// TwinCAT 3 PLC project Fraktal_Tests
// Title: Fraktal_Tests
// Company: fraktal-automation
// Author: fraktal-automation
// ProjectVersion: 0.1.0.10
// Description: Aggregate Fraktal Core + Modules + Press Demo TcUnit gate - excluded from deployed runtime (Core 5.7).
// ProgramVersion: 3.1.4026.24
// libraries:
//   Tc2_Standard, * (Beckhoff Automation GmbH)
//   Tc2_System, * (Beckhoff Automation GmbH)
//   Tc2_Utilities, * (Beckhoff Automation GmbH)
//   Tc3_Module, * (Beckhoff Automation GmbH)
//   Fraktal_Core, 0.25.0.0 (fraktal-automation)
//   Tc2_MC2, * (Beckhoff Automation GmbH)
//   Fraktal_Modules, 0.11.0.3 (fraktal-automation)
//   TcUnit, * (www.tcunit.org)
// project tree:
//   Fraktal_Tests/ FB_ProbeWeeklyLine.TcPOU, FB_Handover_Tests.TcPOU, FB_ProbeRecipeCatalog.TcPOU, PlcTask.TcTTO (not stored), FB_Access_Tests.TcPOU, FB_AlarmLog_Tests.TcPOU (not stored), FB_Base_Tests.TcPOU, FB_ConfigurableCylinderCM_Tests.TcPOU (not stored), FB_ClampEM_Tests.TcPOU, FB_ProbeClampCycle.TcPOU, FB_ProbeClampRoot.TcPOU, FB_UnitTier_Tests.TcPOU, FB_Connector_Tests.TcPOU, FB_CylinderCM_Tests.TcPOU, FB_Decision_Tests.TcPOU, FB_Hmi_Tests.TcPOU, FB_HostEvent_Tests.TcPOU, FB_IoTopologyPublisher_Tests.TcPOU (not stored), FB_InputCM_Tests.TcPOU, FB_ManualCmd_Tests.TcPOU (not stored), FB_MultiRoot_Tests.TcPOU (not stored), FB_Oee_Tests.TcPOU (not stored), FB_PermIntlk_Tests.TcPOU (not stored), FB_PowerGroupCM_Tests.TcPOU (not stored), FB_TwoHandStartCM_Tests.TcPOU (not stored), FB_ConfigWrite_Tests.TcPOU, FB_ProbeConfigPersistence.TcPOU, FB_Shift_Tests.TcPOU, FB_LineData_Tests.TcPOU, FB_ProbeLineSource.TcPOU, FB_ProbeLineUnit.TcPOU, FB_Sha256_Tests.TcPOU, FB_ModelData_Tests.TcPOU, FB_ProbeModelUnit.TcPOU, ST_ProbeModelParCfg.TcDUT, FB_DataClass_Tests.TcPOU, FB_ConfigSet_Tests.TcPOU, FB_ConfigDurability_Tests.TcPOU, FB_ProbeConfigCM.TcPOU, FB_ProbeConfigUnit.TcPOU, FB_ProbeCM.TcPOU, FB_ProbeConnector.TcPOU (not stored), FB_ProbeRaiseChain.TcPOU, FB_ProbeUnitRaise.TcPOU, FB_SequenceRaise_Tests.TcPOU, FB_ProbeLeg.TcPOU, FB_ProbeParChain.TcPOU, FB_ProbeUnitPar.TcPOU, FB_SequencePar_Tests.TcPOU, FB_RobotConnector_Tests.TcPOU, FB_RobotCM_Tests.TcPOU, FB_AxisJog_Tests.TcPOU, FB_Separator_Tests.TcPOU, FB_Engineering_Tests.TcPOU, FB_RobotPlanner_Tests.TcPOU, FB_Separator_Tests.TcPOU, FB_Engineering_Tests.TcPOU, FB_Axis_Tests.TcPOU, FB_Separator_Tests.TcPOU, FB_Engineering_Tests.TcPOU, FB_StateFlag_Tests.TcPOU, FB_ProbeEM.TcPOU (not stored), FB_ProbeUnit.TcPOU, FB_ProbeUnitManual.TcPOU (not stored), FB_Release_Tests.TcPOU (not stored), FB_PartTrace_Tests.TcPOU (not stored), FB_Shelve_Tests.TcPOU, FB_SystemInfrastructure_Tests.TcPOU, FB_TcpDev_Tests.TcPOU (not stored), FB_Timing_Tests.TcPOU, FB_Unit_Tests.TcPOU, FB_ProbeAccessStore.TcPOU, FB_ProbeFileOps.TcPOU, F_ProbeAlarmActive.TcPOU, FB_AccessPersistence_Tests.TcPOU, FB_PlatformHealth_Tests.TcPOU, FB_PersistMedium_Tests.TcPOU, FB_LiveConfig_Tests.TcPOU, PRG_PlatformAcceptance.TcPOU, PRG_TcUnitRunner.TcPOU
// real-time tasks:
//   TASK PlcTask: cycle T#10ms, priority 20, ADS port 350

// ---- Fraktal_Tests/ST_ProbeModelParCfg.TcDUT
// §3.8a probe recipe record: the probe root's own model data.
TYPE ST_ProbeModelParCfg :
STRUCT
    SchemaVersion : UINT := 1;
    Speed         : DINT;
END_STRUCT
END_TYPE

// ---- Fraktal_Tests/FB_ProbeWeeklyLine.TcPOU
FUNCTION_BLOCK FB_ProbeWeeklyLine EXTENDS FB_LineDataV3

Cyclic();

METHOD M_ResetFixture
VAR
    i : INT;
END_VAR
    CalendarV3.SchemaVersion := 3;
    CalendarV3.UtcOffsetMin := 0;
    FOR i := 1 TO PL_Fraktal.MAX_WEEKLY_SHIFTS DO
        CalendarV3.Rows[i].StartMin := -1;
        CalendarV3.Rows[i].DurationMin := 1440;
        CalendarV3.Rows[i].ActiveDays := 0;
        CalendarV3.Rows[i].ProductionTarget := 0;
    END_FOR
END_METHOD

END_FUNCTION_BLOCK

// ---- Fraktal_Tests/FB_Handover_Tests.TcPOU
// AB-to-TC3 portable behavior, exercised in the actual IEC implementation.
FUNCTION_BLOCK FB_Handover_Tests EXTENDS TcUnit.FB_TestSuite
VAR
    _models : FB_ProbeRecipeCatalog;
    _unit : FB_ProbeModelUnit;
    _shift : FB_ProbeConfigUnit;
    _line : FB_ProbeWeeklyLine;
    _schedule : FB_ShiftSchedule;
    _calendar : ST_ShiftCalendarV3;
    _daily : ST_ShiftCalendar;
    _v2 : ST_ShiftCalendarV2;
    _loaded, _default, _a, _b : ST_ProbeModelParCfg;
    _store : FB_LocalConfigStore;
    _info : ST_ConfigSetInfo;
    _record : ST_ConfigRecord;
    _json : FB_ConfigSetJson;
    _init : BOOL;
    _done : ARRAY[1..18] OF BOOL;
    _idx : INT;
    _start, _end : DT;
    _target : UDINT;
    _i : INT;
END_VAR

IF NOT _init THEN
    _init := TRUE;
    _models.M_ResetFixture();
    _default.Speed := 1; _a.Speed := 10; _b.Speed := 20;
    _models.Register(ModelCode := '', RecipeKey := 'ProbeModel', pData := ADR(_default), Size := SIZEOF(_default));
    _models.Register(ModelCode := 'A', RecipeKey := 'ProbeModel', pData := ADR(_a), Size := SIZEOF(_a));
    _models.Register(ModelCode := 'B', RecipeKey := 'ProbeModel', pData := ADR(_b), Size := SIZEOF(_b));
    _unit.ParCfg := _default;
    _unit.Setup(Name := 'Test.Handover', Provider := _models);
    _unit();
    _unit.SetConfigStore(Store := _store);
    FOR _i := 1 TO PL_Fraktal.MAX_CONFIG_SETS DO
        IF _store.M_InfoAt(Index := 1, Info := _info) THEN _store.M_Delete(SetName := _info.SetName); END_IF
    END_FOR
    _line.M_ResetFixture();
    _line.Setup(Name := 'Test.WeeklyLine', LineId := 'handover', Role := E_LineRole.OWNER,
        Source := 0, StaleAfterMs := 0);
    _line();
    _shift.Setup(Name := 'Test.Weekly');
    _shift.SetLine(pLine := ADR(_line));
END_IF
Clone_is_inactive_and_preserves_ordinals();
Duplicate_missing_and_oversize_models_are_atomic();
Clone_rechecks_effective_read_and_write_access();
Complete_model_set_creates_without_running_load();
Current_export_is_immutable_and_uses_no_saved_slot();
Current_export_replay_and_connection_mix_are_refused();
Current_export_rechecks_permissions_and_logout();
Aborted_overwrite_preserves_the_previous_saved_set();
Daily_and_V2_migration_preserve_identity_and_disable_fifth();
Weekly_validation_rejects_overlap_wrap_and_bad_ranges();
Five_rows_select_their_own_weekday_boundaries();
Whole_calendar_transaction_is_atomic();
Off_time_production_and_empty_calendar_edits_are_preserved();
Target_edits_wait_for_boundary_and_history_is_immutable();
Clock_jumps_close_once_without_negative_history();
Manual_OEE_reset_aligns_factors_with_new_count_epoch();
Busy_creation_and_full_catalog_preserve_existing_storage();
Weekly_owner_builds_its_complete_image();

METHOD Clone_is_inactive_and_preserves_ordinals
TEST('Clone_is_inactive_and_preserves_ordinals');
IF NOT _done[1] THEN
AssertTrue(Condition := _unit.CreateModel(ModelCode := 'C', SourceIndex := 2,
    FromSet := FALSE, SetName := ''), Message := 'clone accepted');
AssertEquals_INT(Expected := 3, Actual := _unit.AvailableModelCount, Message := 'appended');
AssertEquals_STRING(Expected := 'A', Actual := _unit.AvailableModels[1].ModelCode, Message := 'ordinal A unchanged');
AssertEquals_STRING(Expected := 'B', Actual := _unit.AvailableModels[2].ModelCode, Message := 'ordinal B unchanged');
AssertEquals_DINT(Expected := 1, Actual := _unit.ParCfg.Speed, Message := 'live recipe unchanged');
AssertTrue(Condition := _models.Load(ModelCode := 'C', RecipeKey := 'ProbeModel',
    pParCfg := ADR(_loaded), Size := SIZEOF(_loaded)), Message := 'provider owns clone');
AssertEquals_DINT(Expected := 20, Actual := _loaded.Speed, Message := 'source model copied');
    _done[1] := TRUE;
END_IF
TEST_FINISHED();
END_METHOD

METHOD Duplicate_missing_and_oversize_models_are_atomic
TEST('Duplicate_missing_and_oversize_models_are_atomic');
IF NOT _done[2] THEN
AssertFalse(Condition := _unit.CreateModel(ModelCode := 'C', SourceIndex := 0, FromSet := FALSE,
    SetName := ''), Message := 'duplicate refused');
AssertFalse(Condition := _unit.CreateModel(ModelCode := 'D', SourceIndex := 99, FromSet := FALSE,
    SetName := ''), Message := 'missing source refused');
AssertFalse(Condition := _unit.CreateModel(ModelCode := 'abcdefghijklmnopqrstuvwxyzabcdefghijklmnopqrstuvwxyzabcdefghijklm',
    SourceIndex := 0, FromSet := FALSE, SetName := ''), Message := '65-byte code refused');
AssertEquals_INT(Expected := 3, Actual := _unit.AvailableModelCount, Message := 'no partial publication');
    _done[2] := TRUE;
END_IF
TEST_FINISHED();
END_METHOD

METHOD Clone_rechecks_effective_read_and_write_access
TEST('Clone_rechecks_effective_read_and_write_access');
IF NOT _done[3] THEN
_unit.M_SetConfigAccess(WriteKey := 'probe.speed', ClassId := '',
    MinReadLevel := E_AccessLevel.ENGINEER, MinWriteLevel := E_AccessLevel.NONE);
AssertFalse(Condition := _unit.CreateModel(ModelCode := 'DeniedRead', SourceIndex := 0,
    FromSet := FALSE, SetName := ''), Message := 'read denied');
_unit.M_SetConfigAccess(WriteKey := 'probe.speed', ClassId := '',
    MinReadLevel := E_AccessLevel.NONE, MinWriteLevel := E_AccessLevel.ENGINEER);
AssertFalse(Condition := _unit.CreateModel(ModelCode := 'DeniedWrite', SourceIndex := 0,
    FromSet := FALSE, SetName := ''), Message := 'write denied');
_unit.M_SetConfigAccess(WriteKey := 'probe.speed', ClassId := '',
    MinReadLevel := E_AccessLevel.NONE, MinWriteLevel := E_AccessLevel.NONE);
AssertEquals_INT(Expected := 3, Actual := _unit.AvailableModelCount, Message := 'denials leave catalog');
    _done[3] := TRUE;
END_IF
TEST_FINISHED();
END_METHOD

METHOD Complete_model_set_creates_without_running_load
TEST('Complete_model_set_creates_without_running_load');
IF NOT _done[4] THEN
AssertTrue(Condition := _unit.SaveConfigSet(SetName := 'model-source', Kind := E_ConfigKind.PAR_CFG),
    Message := 'model snapshot saved');
AssertFalse(Condition := _unit.LoadConfigSet(SetName := 'model-source'), Message := 'running load still refused');
AssertTrue(Condition := _unit.CreateModel(ModelCode := 'FromSet', SourceIndex := 0,
    FromSet := TRUE, SetName := 'model-source'), Message := 'complete Model set creates');
AssertEquals_DINT(Expected := 1, Actual := _unit.ParCfg.Speed, Message := 'running recipe stays');
    _done[4] := TRUE;
END_IF
TEST_FINISHED();
END_METHOD

METHOD Current_export_is_immutable_and_uses_no_saved_slot
TEST('Current_export_is_immutable_and_uses_no_saved_slot');
IF NOT _done[5] THEN
_unit.HmiRequest.Kind := E_HmiRequestKind.EXPORT_CURRENT_CONFIG;
_unit.HmiRequest.TextValue := 'current'; _unit.HmiRequest.NameValue := 'connection-A';
_unit.HmiRequest.IntValue := TO_DINT(E_ConfigKind.PAR_CFG); _unit.HmiRequest.DurationMs := 2;
_unit.HmiRequest.Sequence := _unit.HmiRequest.Sequence + 1; _unit();
AssertTrue(Condition := _unit.HmiResponse.Accepted, Message := 'current header accepted');
_b.Speed := 99; // simulated owner update after capture, no mailbox interleaving
_unit.HmiRequest.Kind := E_HmiRequestKind.EXPORT_CONFIG_SET;
_unit.HmiRequest.IntValue := 1; _unit.HmiRequest.Sequence := _unit.HmiRequest.Sequence + 1; _unit();
AssertTrue(Condition := _unit.HmiResponse.Accepted, Message := 'continuation accepted');
AssertTrue(Condition := _json.M_ParseRecord(Line := _unit.ConfigSetDocument, Record := _record), Message := 'complete JSON record');
AssertEquals_STRING(Expected := '20', Actual := _record.ValueText, Message := 'captured value immutable');
AssertEquals_INT(Expected := 1, Actual := _store.M_Count(), Message := 'no saved slot consumed');
    _done[5] := TRUE;
END_IF
TEST_FINISHED();
END_METHOD

METHOD Current_export_replay_and_connection_mix_are_refused
TEST('Current_export_replay_and_connection_mix_are_refused');
IF NOT _done[6] THEN
AssertTrue(Condition := _unit.ExportCurrentConfig(SetName := 'current', Kind := E_ConfigKind.PAR_CFG,
    ModelIndex := 0, Token := 'connection-A'), Message := 'snapshot opened');
_unit.HmiRequest.Kind := E_HmiRequestKind.EXPORT_CONFIG_SET;
_unit.HmiRequest.NameValue := 'connection-B'; _unit.HmiRequest.TextValue := 'current';
_unit.HmiRequest.IntValue := 1; _unit.HmiRequest.Sequence := _unit.HmiRequest.Sequence + 1; _unit();
AssertFalse(Condition := _unit.HmiResponse.Accepted, Message := 'foreign connection refused');
_unit.HmiRequest.NameValue := 'connection-A'; _unit.HmiRequest.Sequence := _unit.HmiRequest.Sequence + 1; _unit();
AssertFalse(Condition := _unit.HmiResponse.Accepted, Message := 'interrupted cursor cannot replay');
    _done[6] := TRUE;
END_IF
TEST_FINISHED();
END_METHOD

METHOD Current_export_rechecks_permissions_and_logout
TEST('Current_export_rechecks_permissions_and_logout');
IF NOT _done[7] THEN
AssertTrue(Condition := _unit.ExportCurrentConfig(SetName := 'current', Kind := E_ConfigKind.PAR_CFG,
    ModelIndex := 0, Token := 'permission'), Message := 'snapshot opened');
_unit.M_SetConfigAccess(WriteKey := 'probe.speed', ClassId := '',
    MinReadLevel := E_AccessLevel.ADMIN, MinWriteLevel := E_AccessLevel.NONE);
_unit.HmiRequest.Kind := E_HmiRequestKind.EXPORT_CONFIG_SET;
_unit.HmiRequest.NameValue := 'permission'; _unit.HmiRequest.TextValue := 'current';
_unit.HmiRequest.IntValue := 1; _unit.HmiRequest.Sequence := _unit.HmiRequest.Sequence + 1; _unit();
AssertFalse(Condition := _unit.HmiResponse.Accepted, Message := 'read downgrade stops continuation');
AssertEquals_STRING(Expected := '', Actual := _unit.ConfigSetDocument, Message := 'no disclosure');
_unit.M_SetConfigAccess(WriteKey := 'probe.speed', ClassId := '',
    MinReadLevel := E_AccessLevel.NONE, MinWriteLevel := E_AccessLevel.NONE);
AssertTrue(Condition := _unit.ExportCurrentConfig(SetName := 'current', Kind := E_ConfigKind.PAR_CFG,
    ModelIndex := 0, Token := 'logout'), Message := 'second snapshot opened');
_unit.Access.RequestLogout();
_unit.HmiRequest.NameValue := 'logout';
_unit.HmiRequest.Sequence := _unit.HmiRequest.Sequence + 1; _unit();
AssertFalse(Condition := _unit.HmiResponse.Accepted, Message := 'logout invalidates snapshot session');
AssertEquals_STRING(Expected := '', Actual := _unit.ConfigSetDocument, Message := 'pending logout discloses no line');
    _done[7] := TRUE;
END_IF
TEST_FINISHED();
END_METHOD

METHOD Aborted_overwrite_preserves_the_previous_saved_set
TEST('Aborted_overwrite_preserves_the_previous_saved_set');
IF NOT _done[8] THEN
_store.M_ReadInfo(SetName := 'model-source', Info := _info);
_store.M_ReadRecord(SetName := 'model-source', Index := 1, Record := _record);
AssertTrue(Condition := _store.M_SaveBegin(Info := _info), Message := 'overwrite begins');
_record.ValueText := '123'; _store.M_SaveRecord(Record := _record);
_store.M_SaveAbort();
_store.M_ReadRecord(SetName := 'model-source', Index := 1, Record := _record);
AssertEquals_STRING(Expected := '1', Actual := _record.ValueText, Message := 'old set stays byte-valid');
    _done[8] := TRUE;
END_IF
TEST_FINISHED();
END_METHOD

METHOD Daily_and_V2_migration_preserve_identity_and_disable_fifth
TEST('Daily_and_V2_migration_preserve_identity_and_disable_fifth');
IF NOT _done[9] THEN
FOR _i := 1 TO PL_Fraktal.MAX_SHIFTS DO _daily.StartMin[_i] := -1; END_FOR
_daily.UtcOffsetMin := -840; _daily.StartMin[2] := 360;
AssertTrue(Condition := _schedule.M_MigrateV1(Source := _daily, Target := _calendar), Message := 'sole daily row migrates');
AssertEquals_DINT(Expected := 1440, Actual := _calendar.Rows[2].DurationMin, Message := 'sole row 24 hours');
AssertEquals_DINT(Expected := 127, Actual := _calendar.Rows[2].ActiveDays, Message := 'all weekdays');
AssertEquals_DINT(Expected := -1, Actual := _calendar.Rows[5].StartMin, Message := 'fifth unused');
_v2.SchemaVersion := 2; _v2.UtcOffsetMin := 0;
_v2.Rows[4].StartMin := 480; _v2.Rows[4].DurationMin := 720; _v2.Rows[4].ActiveDays := 96;
AssertTrue(Condition := _schedule.M_MigrateV2(Source := _v2, Target := _calendar), Message := 'weekly V2 migrates');
AssertEquals_DINT(Expected := 480, Actual := _calendar.Rows[4].StartMin, Message := 'index four preserved');
AssertEquals_DINT(Expected := 0, Actual := _calendar.Rows[4].ProductionTarget, Message := 'no invented target');
    _done[9] := TRUE;
END_IF
TEST_FINISHED();
END_METHOD

METHOD Weekly_validation_rejects_overlap_wrap_and_bad_ranges
TEST('Weekly_validation_rejects_overlap_wrap_and_bad_ranges');
IF NOT _done[10] THEN
_calendar.SchemaVersion := 3; _calendar.UtcOffsetMin := 0;
FOR _i := 1 TO PL_Fraktal.MAX_WEEKLY_SHIFTS DO
    _calendar.Rows[_i].StartMin := -1; _calendar.Rows[_i].ActiveDays := 0;
    _calendar.Rows[_i].DurationMin := 60; _calendar.Rows[_i].ProductionTarget := 0;
END_FOR
_calendar.Rows[1].StartMin := 1380; _calendar.Rows[1].DurationMin := 120; _calendar.Rows[1].ActiveDays := 64;
_calendar.Rows[2].StartMin := 0; _calendar.Rows[2].DurationMin := 60; _calendar.Rows[2].ActiveDays := 1;
AssertFalse(Condition := _schedule.M_Validate(Calendar := _calendar), Message := 'Sunday wrap overlaps Monday');
_calendar.Rows[2].StartMin := 60;
AssertTrue(Condition := _schedule.M_Validate(Calendar := _calendar), Message := 'half-open adjacency accepted');
_calendar.Rows[2].DurationMin := 0;
AssertFalse(Condition := _schedule.M_Validate(Calendar := _calendar), Message := 'zero duration refused');
_calendar.Rows[2].DurationMin := 60; _calendar.Rows[2].ProductionTarget := -1;
AssertFalse(Condition := _schedule.M_Validate(Calendar := _calendar), Message := 'negative target refused');
    _done[10] := TRUE;
END_IF
TEST_FINISHED();
END_METHOD

METHOD Five_rows_select_their_own_weekday_boundaries
TEST('Five_rows_select_their_own_weekday_boundaries');
IF NOT _done[11] THEN
_calendar.SchemaVersion := 3; _calendar.UtcOffsetMin := 0;
FOR _i := 1 TO PL_Fraktal.MAX_WEEKLY_SHIFTS DO
    _calendar.Rows[_i].StartMin := (_i - 1) * 120; _calendar.Rows[_i].DurationMin := 60;
    _calendar.Rows[_i].ActiveDays := 1; _calendar.Rows[_i].ProductionTarget := _i * 10;
END_FOR
AssertTrue(Condition := _schedule.M_Validate(Calendar := _calendar), Message := 'all five valid');
FOR _i := 1 TO PL_Fraktal.MAX_WEEKLY_SHIFTS DO
    _schedule.M_Interval(Now := UDINT_TO_DT(DT_TO_UDINT(DT#2026-10-05-00:00:00) + TO_UDINT((_i - 1) * 7200)),
        Calendar := _calendar, ShiftIndex => _idx, StartAt => _start, EndAt => _end, Target => _target);
    AssertEquals_INT(Expected := _i, Actual := _idx, Message := 'each slot activates at its own boundary');
    AssertEquals_UDINT(Expected := TO_UDINT(_i * 10), Actual := _target, Message := 'own target');
END_FOR
    _done[11] := TRUE;
END_IF
TEST_FINISHED();
END_METHOD

METHOD Whole_calendar_transaction_is_atomic
TEST('Whole_calendar_transaction_is_atomic');
IF NOT _done[12] THEN
AssertTrue(Condition := _line.M_BeginConfigBatch(), Message := 'calendar batch begins');
_line.M_StageConfigWrite(Scope := 'Test.WeeklyLine', WriteKey := 'line.shift.1.startMin', Revision := 1,
    TextValue := '0', RootReady := TRUE);
_line.M_StageConfigWrite(Scope := 'Test.WeeklyLine', WriteKey := 'line.shift.1.activeDays', Revision := 1,
    TextValue := '127', RootReady := TRUE);
_line.M_StageConfigWrite(Scope := 'Test.WeeklyLine', WriteKey := 'line.shift.2.startMin', Revision := 1,
    TextValue := '0', RootReady := TRUE);
_line.M_StageConfigWrite(Scope := 'Test.WeeklyLine', WriteKey := 'line.shift.2.activeDays', Revision := 1,
    TextValue := '127', RootReady := TRUE);
AssertFalse(Condition := _line.M_CommitConfigBatch(), Message := 'overlapping whole candidate refused');
AssertEquals_DINT(Expected := -1, Actual := _line.CalendarV3.Rows[1].StartMin, Message := 'first field stays unchanged');
    _done[12] := TRUE;
END_IF
TEST_FINISHED();
END_METHOD

METHOD Off_time_production_and_empty_calendar_edits_are_preserved
TEST('Off_time_production_and_empty_calendar_edits_are_preserved');
IF NOT _done[13] THEN
_shift.M_ShiftTick(Now := DT#2026-10-05-00:00:00, Synchronized := TRUE);
FOR _i := 1 TO 7 DO _shift.CountGood(); END_FOR
_line.M_ApplyConfigWrite(Scope := 'Test.WeeklyLine', WriteKey := 'line.shift.1.productionTarget',
    Revision := 1, TextValue := '100', RootReady := TRUE); _line();
AssertFalse(Condition := _shift.M_ShiftTick(Now := DT#2026-10-05-00:01:00, Synchronized := TRUE),
    Message := 'empty schedule edit does not close off production');
AssertEquals_UDINT(Expected := 7, Actual := _shift.GoodCount, Message := 'off production remains');
_line.M_ApplyConfigWrite(Scope := 'Test.WeeklyLine', WriteKey := 'line.shift.1.durationMin',
    Revision := 1, TextValue := '60', RootReady := TRUE);
_line.M_ApplyConfigWrite(Scope := 'Test.WeeklyLine', WriteKey := 'line.shift.1.startMin',
    Revision := 1, TextValue := '0', RootReady := TRUE);
_line.M_ApplyConfigWrite(Scope := 'Test.WeeklyLine', WriteKey := 'line.shift.1.activeDays',
    Revision := 1, TextValue := '127', RootReady := TRUE); _line();
AssertTrue(Condition := _shift.M_ShiftTick(Now := DT#2026-10-05-00:02:00, Synchronized := TRUE),
    Message := 'starting active shift first closes off interval');
AssertEquals_INT(Expected := 0, Actual := _shift.ShiftHistory[1].ShiftIndex, Message := 'off interval identity');
AssertEquals_UDINT(Expected := 7, Actual := _shift.ShiftHistory[1].GoodCount, Message := 'off production archived');
    _done[13] := TRUE;
END_IF
TEST_FINISHED();
END_METHOD

METHOD Target_edits_wait_for_boundary_and_history_is_immutable
TEST('Target_edits_wait_for_boundary_and_history_is_immutable');
IF NOT _done[14] THEN
AssertEquals_UDINT(Expected := 100, Actual := _shift.ShiftProductionTarget, Message := 'target latched at entry');
FOR _i := 1 TO 3 DO _shift.CountGood(); END_FOR
_line.M_ApplyConfigWrite(Scope := 'Test.WeeklyLine', WriteKey := 'line.shift.1.productionTarget',
    Revision := 1, TextValue := '200', RootReady := TRUE); _line();
_shift.M_ShiftTick(Now := DT#2026-10-05-00:30:00, Synchronized := TRUE);
AssertEquals_UDINT(Expected := 100, Actual := _shift.ShiftProductionTarget, Message := 'mid-shift edit deferred');
AssertTrue(Condition := _shift.M_ShiftTick(Now := DT#2026-10-05-01:00:00, Synchronized := TRUE), Message := 'natural end closes');
AssertEquals_UDINT(Expected := 100, Actual := _shift.ShiftHistory[1].ProductionTarget, Message := 'old target in history');
AssertEquals_UDINT(Expected := 0, Actual := _shift.ShiftProductionTarget, Message := 'off target unset');
    _done[14] := TRUE;
END_IF
TEST_FINISHED();
END_METHOD

METHOD Clock_jumps_close_once_without_negative_history
TEST('Clock_jumps_close_once_without_negative_history');
IF NOT _done[15] THEN
FOR _i := 1 TO 2 DO _shift.CountGood(); END_FOR
AssertTrue(Condition := _shift.M_ShiftTick(Now := DT#2026-10-07-00:30:00, Synchronized := TRUE), Message := 'forward jump closes once');
AssertFalse(Condition := _shift.ShiftHistory[1].TimeSynchronized, Message := 'jump quality unverified');
AssertEquals_INT(Expected := 3, Actual := _shift.ShiftHistoryCount, Message := 'no fabricated intervening shifts');
AssertFalse(Condition := _shift.M_ShiftTick(Now := DT#2026-10-06-00:00:00, Synchronized := TRUE), Message := 'backward jump cannot close');
AssertEquals_INT(Expected := 3, Actual := _shift.ShiftHistoryCount, Message := 'history unchanged');
    _done[15] := TRUE;
END_IF
TEST_FINISHED();
END_METHOD

METHOD Manual_OEE_reset_aligns_factors_with_new_count_epoch
TEST('Manual_OEE_reset_aligns_factors_with_new_count_epoch');
IF NOT _done[16] THEN
FOR _i := 1 TO 10 DO _unit.CountGood(); END_FOR
FOR _i := 1 TO 5 DO _unit.CountNok(Reason := E_Reason.TEST_FAULT); END_FOR
AssertTrue(Condition := _unit.ResetOee(), Message := 'manual reset accepted');
AssertFalse(Condition := _unit.Oee.QualValid, Message := 'old counts do not make new quality valid');
AssertEquals_UDINT(Expected := 10, Actual := _unit.GoodCount, Message := 'published production count preserved');
    _done[16] := TRUE;
END_IF
TEST_FINISHED();
END_METHOD

METHOD Busy_creation_and_full_catalog_preserve_existing_storage
VAR
    modelIndex : INT;
    code : STRING(64);
END_VAR
TEST('Busy_creation_and_full_catalog_preserve_existing_storage');
IF NOT _done[17] THEN
AssertTrue(Condition := _unit.Start(), Message := 'probe starts its continuous command');
_unit();
AssertTrue(Condition := _unit.Busy, Message := 'creation fixture is actually BUSY');
FOR modelIndex := _unit.AvailableModelCount + 1 TO _unit.ModelCapacity DO
    code := CONCAT('Catalog', INT_TO_STRING(modelIndex));
    AssertTrue(Condition := _unit.CreateModel(ModelCode := code, SourceIndex := 1,
        FromSet := FALSE, SetName := ''), Message := 'inactive append permitted while BUSY');
END_FOR
AssertFalse(Condition := _unit.CreateModel(ModelCode := 'Overflow', SourceIndex := 1,
    FromSet := FALSE, SetName := ''), Message := 'full catalog refuses atomically');
AssertEquals_INT(Expected := _unit.ModelCapacity, Actual := _unit.AvailableModelCount,
    Message := 'full publication has exact capacity');
AssertTrue(Condition := _models.Load(ModelCode := 'A', RecipeKey := 'ProbeModel',
    pParCfg := ADR(_loaded), Size := SIZEOF(_loaded)), Message := 'original address remains available');
AssertEquals_DINT(Expected := 10, Actual := _loaded.Speed, Message := 'original seed bytes unchanged');
AssertEquals_DINT(Expected := 1, Actual := _unit.ParCfg.Speed, Message := 'live recipe remains unchanged');
AssertTrue(Condition := _unit.Busy, Message := 'creation does not stop running command');
    _done[17] := TRUE;
END_IF
TEST_FINISHED();
END_METHOD

METHOD Weekly_owner_builds_its_complete_image
VAR
    rowIndex : INT;
    fifthPresent : BOOL;
END_VAR
TEST('Weekly_owner_builds_its_complete_image');
IF NOT _done[18] THEN
_line();
AssertEquals_INT(Expected := 21, Actual := _line.Image.Count,
    Message := 'cyclic owner publication includes every weekly calendar capability');
FOR rowIndex := 1 TO _line.Image.Count DO
    IF _line.Image.Records[rowIndex].WriteKey = 'line.shift.5.productionTarget' THEN
        fifthPresent := TRUE;
    END_IF
END_FOR
AssertTrue(Condition := fifthPresent, Message := 'fifth target is in the owner image');
    _done[18] := TRUE;
END_IF
TEST_FINISHED();
END_METHOD

END_FUNCTION_BLOCK

// ---- Fraktal_Tests/FB_ProbeRecipeCatalog.TcPOU
FUNCTION_BLOCK FB_ProbeRecipeCatalog EXTENDS FB_LocalRecipeProvider

;

METHOD M_ResetFixture
// This seam belongs only to the isolated TcUnit image, never production.
_catalog.SchemaVersion := 1;
_catalog.Count := 0;
_catalogInitialized := FALSE;
_catalogRestoreVersion := 0;
_n := 0;
END_METHOD

END_FUNCTION_BLOCK

// ---- Fraktal_Tests/FB_ProbeModelUnit.TcPOU
// §3.8a probe root: one model-data value in its own recipe record (registered
// as model data) and one station value beside it, over two catalog models.
FUNCTION_BLOCK FB_ProbeModelUnit EXTENDS FB_UnitBase
VAR_INPUT
    ParCfg : ST_ProbeModelParCfg;
    StationLimit : DINT := 5;
END_VAR

Cyclic();

METHOD Setup : BOOL
VAR_INPUT
    Name     : STRING(80);
    Provider : I_RecipeProvider;
END_VAR
VAR
    model : ST_ModelId;
END_VAR
_M_SetName(Name);
StallTime := T#0S;
Setup := M_RegisterConfigNumber(Key := 'probe.speed', Item := 'ParCfg/Speed',
    LabelKey := 'project.test.speed', Unit := E_EngUnit.NONE,
    Kind := E_ConfigKind.PAR_CFG, Storage := E_ConfigStorage.AS_DINT,
    pTarget := ADR(ParCfg.Speed), Minimum := 0.0, Maximum := 1000.0,
    RequiresReady := FALSE);
Setup := M_RegisterConfigNumber(Key := 'probe.limit', Item := 'StationCfg/Limit',
    LabelKey := 'project.test.limit', Unit := E_EngUnit.NONE,
    Kind := E_ConfigKind.STATION_CFG, Storage := E_ConfigStorage.AS_DINT,
    pTarget := ADR(StationLimit), Minimum := 0.0, Maximum := 100.0,
    RequiresReady := FALSE) AND Setup;
Setup := M_RegisterModelData(pData := ADR(ParCfg), Size := SIZEOF(ParCfg),
    RecipeKey := 'ProbeModel', Provider := Provider) AND Setup;
model.ModelCode := 'A';
Setup := RegisterAvailableModel(Id := model) AND Setup;
model.ModelCode := 'B';
Setup := RegisterAvailableModel(Id := model) AND Setup;
END_METHOD

METHOD PROTECTED _M_Dispatch
_M_SetStep(StepNo := 100, StepName := 'project.test.stepA', Awaits := 0,
    AwaitingLabel := '', TimeClass := E_TimeClass.WORK, ExpectedTime := T#0S);
END_METHOD

END_FUNCTION_BLOCK

// ---- Fraktal_Tests/FB_ProbeConfigUnit.TcPOU
// §3.8b probe root: one own editable value plus one child that owns three more.
// The point of the pair is the walk — the root registers no routing code at all,
// so a test that writes a child's value proves the generic path rather than a
// hand-written override (§1.1 O1).
FUNCTION_BLOCK FB_ProbeConfigUnit EXTENDS FB_UnitBase
VAR_OUTPUT
    Child : FB_ProbeConfigCM;
END_VAR
VAR_INPUT
    CycleLimit : DINT := 100;
END_VAR

Cyclic();

METHOD Setup : BOOL
VAR_INPUT
    Name : STRING(80);
END_VAR
_M_SetName(Name);
StallTime := T#0S;
Setup := M_RegisterConfigNumber(Key := 'probe.cycleLimit',
    Item := 'StationCfg/CycleLimit', LabelKey := 'project.test.cycleLimit',
    Unit := E_EngUnit.NONE, Kind := E_ConfigKind.STATION_CFG,
    Storage := E_ConfigStorage.AS_DINT, pTarget := ADR(CycleLimit),
    Minimum := 1.0, Maximum := 1000.0, RequiresReady := FALSE);
Setup := Child.Setup(Name := CONCAT(Name, '.Child')) AND Setup;
IF Setup THEN
    Setup := _M_Register(Child);
END_IF
END_METHOD

METHOD PROTECTED _M_Dispatch
_M_SetStep(StepNo := 100, StepName := 'project.test.stepA', Awaits := 0,
    AwaitingLabel := '', TimeClass := E_TimeClass.WORK, ExpectedTime := T#0S);
END_METHOD

// Test seam. The child is reachable from outside for READING, but a nested FB
// behind an output is not an assignment target, so the owner sets it — which is
// also how a real composite would configure its own child.
METHOD M_SetChildRefuse
VAR_INPUT
    Text : STRING(255);
END_VAR
Child.RefuseText := Text;
END_METHOD

END_FUNCTION_BLOCK

// ---- Fraktal_Tests/FB_ProbeConfigCM.TcPOU
// §3.8b probe: a leaf module that declares one editable value of each storage
// class, so the registry can be tested where it actually lives — on a child,
// reached by the root's recursive walk rather than by the root's own handler.
// Values are plain VAR_INPUT here (configuration data, per the transport
// contract): this suite proves registration, validation and routing, while
// retention is TwinCAT's job and is not what these tests assert.
FUNCTION_BLOCK FB_ProbeConfigCM EXTENDS FB_ControlModuleBase
VAR_INPUT
    SettleTime : TIME := T#500MS;
    Retries    : DINT := 3;
    Enabled    : BOOL := TRUE;
    Label      : STRING(80) := 'default';
    Mode       : DINT := 1;              // an enumeration stored as its ordinal
    // Test seam for the module-invariant hook: the one candidate this module
    // refuses whatever its type and range say.
    RefuseText : STRING(255);
END_VAR
VAR_OUTPUT
    RefusedCount : UDINT;            // proves the hook ran, not just that a write failed
END_VAR

Cyclic();

METHOD Setup : BOOL
VAR_INPUT
    Name : STRING(80);
END_VAR
_M_SetName(Name);
Setup := M_RegisterConfigDuration(Key := 'probe.settleTime',
    Item := 'StationCfg/SettleTime', LabelKey := 'project.test.settleTime',
    Kind := E_ConfigKind.STATION_CFG, pTarget := ADR(SettleTime),
    MinimumMs := 0, MaximumMs := 5000, RequiresReady := TRUE);
Setup := M_RegisterConfigNumber(Key := 'probe.retries',
    Item := 'StationCfg/Retries', LabelKey := 'project.test.retries', Unit := E_EngUnit.NONE,
    Kind := E_ConfigKind.STATION_CFG, Storage := E_ConfigStorage.AS_DINT,
    pTarget := ADR(Retries), Minimum := 0.0, Maximum := 10.0,
    RequiresReady := FALSE) AND Setup;
Setup := M_RegisterConfigFlag(Key := 'probe.enabled',
    Item := 'StationCfg/Enabled', LabelKey := 'project.test.enabled',
    Kind := E_ConfigKind.STATION_CFG, pTarget := ADR(Enabled),
    RequiresReady := FALSE) AND Setup;
Setup := M_RegisterConfigWrite(Key := 'probe.label',
    Item := 'StationCfg/Label', Revision := 2, Kind := E_ConfigKind.STATION_CFG,
    ValueType := E_ConfigValueType.TEXT, Storage := E_ConfigStorage.AS_STRING,
    pTarget := ADR(Label), RequiresReady := FALSE, HasMinimum := FALSE,
    HasMaximum := FALSE, Minimum := 0.0, Maximum := 0.0, Unit := E_EngUnit.NONE,
    LabelKey := 'project.test.label', MaxLength := 80,
    EnumDomain := '', EnumLabelKey := '') AND Setup;
Setup := M_RegisterConfigChoice(Key := 'probe.mode', Item := 'StationCfg/Mode',
    LabelKey := 'project.test.mode', Kind := E_ConfigKind.STATION_CFG,
    Storage := E_ConfigStorage.AS_DINT, pTarget := ADR(Mode), Domain := '0|1|2',
    EnumLabelKey := 'project.test.modeValue', RequiresReady := FALSE) AND Setup;
END_METHOD

METHOD PROTECTED _M_Dispatch
_M_Complete();
END_METHOD

// §3.10.2 — the module-specific invariant hook. Refuses one candidate outright
// so the suite can prove a hook rejection leaves the value untouched, exactly
// like a range rejection does.
METHOD PROTECTED _M_OnConfigWrite : BOOL
VAR_INPUT
    WriteKey  : STRING(160);
    TextValue : STRING(255);
END_VAR
_M_OnConfigWrite := SUPER^._M_OnConfigWrite(WriteKey := WriteKey,
    TextValue := TextValue);
IF (RefuseText <> '') AND (TextValue = RefuseText) THEN
    RefusedCount := RefusedCount + 1;
    _M_OnConfigWrite := FALSE;
END_IF
END_METHOD

END_FUNCTION_BLOCK

// ---- Fraktal_Tests/FB_Access_Tests.TcPOU
// Core §7.7 under test: open-by-default, threshold denial, data-driven login through
// the local provider, secret cleared, logout re-denies, denied attempts audited.
FUNCTION_BLOCK FB_Access_Tests EXTENDS TcUnit.FB_TestSuite
VAR
    _u  : FB_ProbeUnit;
    _pr : FB_LocalAccessProvider;
    _w  : BOOL;
END_VAR

Default_policy_is_fully_open();
Threshold_denies_then_login_permits_then_logout_denies();
Policy_rejects_invalid_ordinals_and_timeout();
Re_registering_replaces_the_PIN();

METHOD Default_policy_is_fully_open
TEST('Default_policy_is_fully_open');
IF NOT _w THEN
    _u.Setup('Test.AccessUnit');
    // Not under test here: a volatile table, so no previous run's file is a precondition.
    _pr.M_UseKey(Key := '');
    _pr.Register(User := 'tech1', Pin := '4711', Level := E_AccessLevel.TECHNICIAN);
    _u();                                              // first scan wires audit log
    _u.Access.Setup(Provider := _pr, pAlarmLog := ADR(_u.AlarmLog));
    _w := TRUE;
END_IF
AssertTrue(Condition := _u.Access.Permits(Gate := E_GatedAction.MODE_CHANGE),
           Message := 'NONE thresholds: no login needed (7.7b — the fully-open station)');
AssertTrue(Condition := _u.SetMode(Mode := E_Mode.MANUAL),
           Message := 'mode change works without any session');
AssertTrue(Condition := _u.SetMode(Mode := E_Mode.AUTO), Message := 'back to AUTO');
_u(); _u(); _u();
TEST_FINISHED();
END_METHOD

METHOD Threshold_denies_then_login_permits_then_logout_denies
TEST('Threshold_denies_then_login_permits_then_logout_denies');
_u.Access.ConfigureRequired(Gate := E_GatedAction.MODE_CHANGE, Level := E_AccessLevel.TECHNICIAN);
AssertFalse(Condition := _u.SetMode(Mode := E_Mode.MANUAL),
            Message := 'denied below threshold (7.7c) — PLC re-checks, not the HMI');
AssertTrue(Condition := _u.AlarmLog.RingHead > 0,
           Message := 'denied attempt audited as a MESSAGE event (8.3)');
// wrong PIN
_u.Access.RequestLogin(User := 'tech1', Secret := '0000');
_u();
AssertTrue(Condition := _u.Access.LoginFailed, Message := 'wrong PIN rejected');
AssertEquals_DINT(Expected := TO_DINT(E_AccessLevel.NONE),
                  Actual := TO_DINT(_u.Access.CurrentLevel), Message := 'level stays NONE');
// correct PIN — data-driven login (3.10a')
_u.Access.RequestLogin(User := 'tech1', Secret := '4711');
_u();
AssertEquals_DINT(Expected := TO_DINT(E_AccessLevel.TECHNICIAN),
                  Actual := TO_DINT(_u.Access.CurrentLevel), Message := 'TECHNICIAN session');
AssertEquals_STRING(Expected := '', Actual := _u.Access.ReqSecret,
                    Message := 'secret cleared after the attempt (7.7c)');
AssertTrue(Condition := _u.SetMode(Mode := E_Mode.MANUAL),
           Message := 'permitted at sufficient level');
_u.Access.RequestLogout();
_u();
AssertEquals_DINT(Expected := TO_DINT(E_AccessLevel.NONE),
                  Actual := TO_DINT(_u.Access.CurrentLevel), Message := 'logged out');
AssertFalse(Condition := _u.SetMode(Mode := E_Mode.AUTO),
            Message := 'denied again after logout');
_u.Access.ConfigureRequired(Gate := E_GatedAction.MODE_CHANGE, Level := E_AccessLevel.NONE);  // restore
_u.SetMode(Mode := E_Mode.AUTO);
_u(); _u();
TEST_FINISHED();
END_METHOD

METHOD Policy_rejects_invalid_ordinals_and_timeout
VAR
    invalidGate : E_GatedAction;
    invalidLevel : E_AccessLevel;
END_VAR
TEST('Policy_rejects_invalid_ordinals_and_timeout');
invalidGate := 99;
invalidLevel := 99;
AssertFalse(Condition := _u.Access.ConfigureRequired(
    Gate := invalidGate, Level := E_AccessLevel.ADMIN),
    Message := 'out-of-range gate fails closed');
AssertFalse(Condition := _u.Access.ConfigureRequired(
    Gate := E_GatedAction.DATA_WRITE, Level := invalidLevel),
    Message := 'out-of-range level fails closed');
AssertFalse(Condition := _u.Access.ConfigureSessionTimeout(TimeoutMs := 604800001),
    Message := 'timeout above seven days rejected');
AssertTrue(Condition := _u.Access.ConfigureSessionTimeout(TimeoutMs := 900000),
    Message := 'bounded timeout accepted');
AssertEquals_DINT(Expected := 900000,
    Actual := TIME_TO_DINT(_u.Access.Policy.SessionTimeout),
    Message := 'accepted timeout stored in policy');
_u.Access.ConfigureSessionTimeout(TimeoutMs := 0);
TEST_FINISHED();
END_METHOD

// §14 - the table holds only a salted hash, so the PIN is checked by hashing the
// attempt: the new PIN is accepted, the old one and the hash's own inputs are not.
METHOD Re_registering_replaces_the_PIN
VAR
    p : FB_LocalAccessProvider;
END_VAR
TEST('Re_registering_replaces_the_PIN');
AssertTrue(Condition := p.Register(User := 'op', Pin := '1111', Level := E_AccessLevel.OPERATOR),
    Message := 'registered');
AssertTrue(Condition := p.Register(User := 'eng', Pin := '1111', Level := E_AccessLevel.ENGINEER),
    Message := 'a second user may share the PIN (own salt)');
AssertEquals_DINT(Expected := TO_DINT(E_AccessLevel.OPERATOR),
    Actual := TO_DINT(p.Authenticate(User := 'op', Secret := '1111')), Message := 'op accepted');
AssertEquals_DINT(Expected := TO_DINT(E_AccessLevel.ENGINEER),
    Actual := TO_DINT(p.Authenticate(User := 'eng', Secret := '1111')), Message := 'eng accepted');
AssertTrue(Condition := p.Register(User := 'op', Pin := '2222', Level := E_AccessLevel.OPERATOR),
    Message := 're-registered');
AssertEquals_DINT(Expected := TO_DINT(E_AccessLevel.NONE),
    Actual := TO_DINT(p.Authenticate(User := 'op', Secret := '1111')), Message := 'old PIN refused');
AssertEquals_DINT(Expected := TO_DINT(E_AccessLevel.OPERATOR),
    Actual := TO_DINT(p.Authenticate(User := 'op', Secret := '2222')), Message := 'new PIN accepted');
AssertEquals_DINT(Expected := TO_DINT(E_AccessLevel.NONE),
    Actual := TO_DINT(p.Authenticate(User := 'nobody', Secret := '2222')), Message := 'unknown user refused');
AssertEquals_DINT(Expected := TO_DINT(E_AccessLevel.NONE),
    Actual := TO_DINT(p.Authenticate(User := 'op', Secret := '')), Message := 'empty secret refused');
TEST_FINISHED();
END_METHOD

END_FUNCTION_BLOCK

// ---- Fraktal_Tests/FB_ProbeUnit.TcPOU
// minimal Unit for the base suite: 2-step looping chain, one wait-classed step
FUNCTION_BLOCK FB_ProbeUnit EXTENDS FB_UnitBase
VAR_INPUT
    SimA, SimB : BOOL;
    SimFault : BOOL;                    // deterministic fault injection for base-path tests
END_VAR
VAR_OUTPUT
    ModeChangedCount : UDINT;
    ModeExitCount : UDINT;
    ModeExitFirstCount : UDINT;
    LastNewMode : E_Mode;
    LastOldMode : E_Mode;
    LastRequestedMode : E_Mode;
END_VAR

Cyclic();

METHOD Setup : BOOL
VAR_INPUT
    Name : STRING(80);
END_VAR
_M_SetName(Name);
StallTime := T#0S;                       // test: stall pending fires immediately
Setup := TRUE;
END_METHOD

METHOD PROTECTED _M_Dispatch
CASE _step OF
    10:
        _M_SetStep(StepNo := 100, StepName := 'project.test.stepA', Awaits := 0,
            AwaitingLabel := '', TimeClass := E_TimeClass.WORK, ExpectedTime := T#0S);
        IF SimFault THEN
            _M_Fault(E_Reason.TEST_FAULT, 'forced Unit fault');
        ELSIF SimA THEN
            _step := 20;
        END_IF
    20:
        _M_SetStep(StepNo := 200, StepName := 'project.test.stepB', Awaits := 0,
            AwaitingLabel := '', TimeClass := E_TimeClass.WAIT_UPSTREAM, ExpectedTime := T#0S);
        IF SimB THEN
            _step := 30;
        END_IF
    30:
        IF _M_EndOfCycle() THEN
            _step := 10;
        END_IF
ELSE
    _M_Fault(E_Reason.STEP_STALLED, 'undefined step');
END_CASE
END_METHOD

// Test-probe seam for the protected §6.11 host service.
METHOD M_TestAskDecision : BOOL
VAR_INPUT
    Req : ST_DecisionRequest;
END_VAR
_M_AskDecision(Req := Req);
M_TestAskDecision := Decision.Prompt = Req.Prompt;
END_METHOD

METHOD M_TestClearDecision
M_SequenceClearDecision();
END_METHOD

METHOD M_TestTakeDecision : INT
M_TestTakeDecision := _M_TakeDecision();
END_METHOD

METHOD PROTECTED OnModeChanged : DINT
VAR_INPUT
    NewMode : E_Mode;
    OldMode : E_Mode;
END_VAR
OnModeChanged := SUPER^.OnModeChanged(
    NewMode := NewMode, OldMode := OldMode);
ModeChangedCount := ModeChangedCount + 1;
LastNewMode := NewMode;
LastOldMode := OldMode;
END_METHOD

METHOD PROTECTED OnModeExit : DINT
VAR_INPUT
    FirstCall : BOOL;
    RequestedMode : E_Mode;
END_VAR
// This probe wants the default immediate cancel, so the base call is intentional.
OnModeExit := SUPER^.OnModeExit(
    FirstCall := FirstCall, RequestedMode := RequestedMode);
ModeExitCount := ModeExitCount + 1;
IF FirstCall THEN
    ModeExitFirstCount := ModeExitFirstCount + 1;
END_IF
LastRequestedMode := RequestedMode;
END_METHOD

END_FUNCTION_BLOCK

// ---- Fraktal_Tests/FB_Base_Tests.TcPOU
// Base-class TcUnit suite — conformance rows T1/T2/T4 proven ONCE for every
// inheriting type (Core §5.7), plus the EM rollup (T6 at base level).
FUNCTION_BLOCK FB_Base_Tests EXTENDS TcUnit.FB_TestSuite
VAR
    _p1 : FB_ProbeCM;   // T1
    _p2 : FB_ProbeCM;   // T2
    _p4 : FB_ProbeCM;   // T4
    _em : FB_ProbeEM;   // T6 (base-level rollup)
    _d  : ST_Diagnostic;
    _w1, _w2, _w4, _w6 : BOOL;
END_VAR

T1_Handshake_and_execute_drop_reset();
T2_First_out_reason_and_source_path();
T4_Abort_reports_and_no_auto_resume();
T6_Rollup_adopts_child_first_out();

METHOD T1_Handshake_and_execute_drop_reset
TEST('T1_Handshake_and_execute_drop_reset');
IF NOT _w1 THEN
    _p1.Setup('Test.Probe1');
    _w1 := TRUE;
END_IF
_p1.Execute := TRUE;
_p1();
AssertTrue(Condition := _p1.Busy, Message := 'Busy on Execute rising edge');
AssertEquals_UDINT(Expected := 1, Actual := _p1.CommandStarts,
    Message := 'OnCommandStart runs once on the accepted edge');
_p1.SimDone := TRUE;
_p1();
AssertTrue(Condition := _p1.Done,  Message := 'Done on completion');
AssertFalse(Condition := _p1.Busy, Message := 'not Busy when Done');
AssertEquals_UDINT(Expected := 1, Actual := _p1.CommandStarts,
    Message := 'OnCommandStart is not repeated while Execute remains high');
_p1.Execute := FALSE;
_p1.SimDone := FALSE;
_p1();
AssertFalse(Condition := _p1.Busy OR _p1.Done OR _p1.Error OR _p1.Aborted,
            Message := 'idle after Execute drops (Core 6.1 reset)');
_p1.Execute := TRUE;
_p1();
AssertEquals_UDINT(Expected := 2, Actual := _p1.CommandStarts,
    Message := 'a later accepted command gets a fresh start callback');
_p1.SimDone := TRUE;
_p1();
_p1.Execute := FALSE;
_p1();
TEST_FINISHED();
END_METHOD

METHOD T2_First_out_reason_and_source_path
TEST('T2_First_out_reason_and_source_path');
IF NOT _w2 THEN
    _p2.Setup('Test.Probe2');
    _w2 := TRUE;
END_IF
_p2.Execute  := TRUE;
_p2.SimFault := TRUE;
_p2();
AssertTrue(Condition := _p2.Error, Message := 'Error on forced fault');
AssertEquals_DWORD(Expected := TO_DWORD(E_Reason.TEST_FAULT),
                   Actual   := _p2.ErrorID,
                   Message  := 'ErrorID carries the first-out ReasonCode (Core 8.8)');
_d := _p2.GetFaultSummary();
AssertEquals_STRING(Expected := 'Test.Probe2',
                    Actual   := _d.SourcePath,
                    Message  := 'first-out names the source path (Core 6.9)');
TEST_FINISHED();
END_METHOD

METHOD T4_Abort_reports_and_no_auto_resume
TEST('T4_Abort_reports_and_no_auto_resume');
IF NOT _w4 THEN
    _p4.Setup('Test.Probe4');
    _w4 := TRUE;
END_IF
_p4.Execute := TRUE;
_p4();
AssertTrue(Condition := _p4.Busy, Message := 'Busy before abort');
_p4.Abort := TRUE;
_p4();
AssertTrue(Condition := _p4.Aborted, Message := 'Aborted reported');
_p4.Abort := FALSE;
_p4();
AssertFalse(Condition := _p4.Busy,
            Message := 'no self-resume while Execute stays held (Core 6.1/9.3)');
_p4.Execute := FALSE;
_p4();
AssertFalse(Condition := _p4.Aborted, Message := 'idle after Execute drops');
TEST_FINISHED();
END_METHOD

METHOD T6_Rollup_adopts_child_first_out
TEST('T6_Rollup_adopts_child_first_out');
IF NOT _w6 THEN
    _em.Setup('Test.EM');
    _w6 := TRUE;
END_IF
_em.TestSetChildren(ChildADone := TRUE, ChildAFault := FALSE,
                    ChildBDone := FALSE, ChildBFault := TRUE);
_em.Execute := TRUE;
_em();                          // scan 1: EM Busy, commands children
_em();                          // scan 2: children ran, EM joins/rolls up
_em();                          // scan 3: settle
AssertTrue(Condition := _em.Error, Message := 'EM faults on child error');
_d := _em.GetFaultSummary();
AssertEquals_DWORD(Expected := TO_DWORD(E_Reason.TEST_FAULT),
                   Actual   := TO_DWORD(_d.ReasonCode),
                   Message  := 'EM adopts the child reason verbatim (Core 8.2)');
AssertEquals_STRING(Expected := 'Test.EM.ChildB',
                    Actual   := _d.SourcePath,
                    Message  := 'rollup names the CHILD source path, not the EM');
TEST_FINISHED();
END_METHOD

END_FUNCTION_BLOCK

// ---- Fraktal_Tests/FB_ProbeCM.TcPOU
// Minimal concrete probe for the base classes (Fraktal_QuickStart_and_Suite.md §1).
// Its process logic is only _M_Dispatch. CommandStarts observes the inherited
// command-start callback so the base suite can prove its one-shot semantics.
FUNCTION_BLOCK FB_ProbeCM EXTENDS FB_ControlModuleBase
VAR_INPUT
    SimDone  : BOOL;
    SimFault : BOOL;
    SimState : BOOL;                 // §3.12 the derived fact this probe publishes
    SimPublish : BOOL := TRUE;       // stop publishing to exercise the stale path
END_VAR
VAR_OUTPUT
    CommandStarts : UDINT;
    StateProbe : BOOL;               // what _M_State returned, so the call reads as an assignment
END_VAR

Cyclic();

METHOD Setup : BOOL
VAR_INPUT
    Name : STRING(80);
END_VAR
_M_SetName(Name);
Setup := TRUE;
END_METHOD

METHOD PROTECTED OnCyclic : DINT
OnCyclic := SUPER^.OnCyclic();   // base first (Core §3.14.2)
// §3.12 — a derived flag is published UNCONDITIONALLY every scan. SimPublish exists
// only so the suite can prove what happens when a project breaks that rule.
IF SimPublish THEN
    StateProbe := _M_State(Idx := 1, Key := 'project.test.probeState', Ok := SimState);
END_IF
END_METHOD

METHOD PROTECTED _M_Dispatch
_M_TagCommand(Id := 1, Label := 'PROBE');   // §8.11.4(a) — the one-line command tag
IF SimFault THEN
    _M_Fault(E_Reason.TEST_FAULT, 'probe fault');
ELSIF SimDone THEN
    _M_Complete();
END_IF
END_METHOD

METHOD PROTECTED OnCommandStart : DINT
OnCommandStart := SUPER^.OnCommandStart();
CommandStarts := CommandStarts + 1;
END_METHOD

END_FUNCTION_BLOCK

// ---- Fraktal_Tests/FB_ClampEM_Tests.TcPOU
// Annex H §H.5 — the Composite (EM) tier suite.
//
// §5.7 coverage for this type. Rows T1/T4 and the T2/T6 *mechanisms* are proven
// once in the framework base suite (FB_Base_Tests) and are deliberately NOT
// re-tested here — "verification, like standardization, is paid once at the level
// that owns the behaviour". What this suite owes is the applicable rows re-proven
// with the TYPE's OWN reasons and source paths:
//   T2  first-out carries this type's reason + its own child path  (via T6 case)
//   T3  interlock withholds the output, with this type's path
//   T5  invalid ParCfg -> RECIPE_INVALID, never mis-runs
//   T6  cross-tier rollup: child first-out adopted verbatim  (composite row)
FUNCTION_BLOCK FB_ClampEM_Tests EXTENDS TcUnit.FB_TestSuite
VAR
    _em : FB_ClampEM;
    _hA, _hB : ST_CylinderHal;
    _simA : FB_CylinderSim;
    _pr : FB_LocalRecipeProvider;
    _bCyl : ST_CylinderParCfg;
    _bClamp : ST_ClampParCfg;
    _d : ST_Diagnostic;
    _w : BOOL;
    _i : INT;

    // T3 — a second EM whose CylA permissive is dropped before the command. It needs
    // its OWN cylinder recipe and plant: the shared record sets MoveTimeout := T#0S,
    // so the UNinterlocked partner used to time out in the same scan and the rollup
    // named CylA only because it happened to be first in registration order. With a
    // travel timeout the partner cannot expire, so this test now depends on the
    // interlock alone — and the sims let the suspended clamp finish after it returns.
    _emIntlk : FB_ClampEM;
    _hIA, _hIB : ST_CylinderHal;
    _simIntlkA, _simIntlkB : FB_CylinderSim;
    _prIntlk : FB_LocalRecipeProvider;
    _bCylTravel : ST_CylinderParCfg;

    // T5 — a third EM built on a recipe whose stored ClampEM schema is wrong.
    _emBad : FB_ClampEM;
    _hBA, _hBB : ST_CylinderHal;
    _prBad : FB_LocalRecipeProvider;
    _bClampBad : ST_ClampParCfg;
END_VAR

IF NOT _w THEN
    _bCyl.MoveTimeout := T#0S;               // CylB times out deterministically
    _bClamp.SettleTime := T#0S;
    _pr.Register(ModelCode := '', RecipeKey := 'CylinderCM', pData := ADR(_bCyl), Size := SIZEOF(_bCyl));
    _pr.Register(ModelCode := '', RecipeKey := 'ClampEM', pData := ADR(_bClamp), Size := SIZEOF(_bClamp));
    _em.Setup(Name := 'ClampStation', HalA := _hA, HalB := _hB, Recipe := _pr);
    _simA.Setup(HalRef := _hA, TravelTime := T#0S);
    _bCylTravel.MoveTimeout := T#5S;         // cannot expire inside a test scan
    _prIntlk.Register(ModelCode := '', RecipeKey := 'CylinderCM', pData := ADR(_bCylTravel), Size := SIZEOF(_bCylTravel));
    _prIntlk.Register(ModelCode := '', RecipeKey := 'ClampEM', pData := ADR(_bClamp), Size := SIZEOF(_bClamp));
    _emIntlk.Setup(Name := 'ClampIntlk', HalA := _hIA, HalB := _hIB, Recipe := _prIntlk);
    _simIntlkA.Setup(HalRef := _hIA, TravelTime := T#0S);
    _simIntlkB.Setup(HalRef := _hIB, TravelTime := T#0S);
    // Stored ClampEM record declares schema 2 while the type expects 1 (§3.8).
    _bClampBad.SchemaVersion := 2;
    _prBad.Register(ModelCode := '', RecipeKey := 'CylinderCM', pData := ADR(_bCyl), Size := SIZEOF(_bCyl));
    _prBad.Register(ModelCode := '', RecipeKey := 'ClampEM', pData := ADR(_bClampBad), Size := SIZEOF(_bClampBad));
    _w := TRUE;
END_IF
Clamp_rolls_up_CylB_first_out();
T3_interlock_withholds_child_output();
T5_recipe_schema_mismatch_faults();

METHOD Clamp_rolls_up_CylB_first_out
TEST('Clamp_rolls_up_CylB_first_out');
_em.Command := E_ClampCommand.CLAMP;
_em.Execute := TRUE;
FOR _i := 1 TO 6 DO
    _em();                                   // EM ticks children in OnCyclic
    _simA();                                 // plant completes CylA; CylB never arrives
END_FOR
AssertTrue(Condition := _em.Error, Message := 'EM faults on child error');
_d := _em.GetFaultSummary();
AssertEquals_DWORD(Expected := TO_DWORD(PL_ModuleReasons.CYL_NOT_EXTENDED),
                   Actual   := TO_DWORD(_d.ReasonCode),
                   Message  := 'EM adopts the child first-out verbatim (8.2)');
AssertEquals_STRING(Expected := 'ClampStation.CylB', Actual := _d.SourcePath,
                    Message := 'rollup names CylB, not the EM (H.5)');
TEST_FINISHED();
END_METHOD

// §5.7 T3 for the composite tier: a dropped permissive on a child must withhold
// the physical output and surface the interlock reason THROUGH the EM, naming the
// child that is actually blocked (not the EM) — the composite tier's own
// path/reason pairing, which the base-suite mechanism test cannot assert.
METHOD T3_interlock_withholds_child_output
TEST('T3_interlock_withholds_child_output');
_emIntlk.CylA.SetAreaSafe(Ok := FALSE, DescriptionKey := '');   // the real §7.2 path
_emIntlk.Command := E_ClampCommand.CLAMP;
_emIntlk.Execute := TRUE;
FOR _i := 1 TO 4 DO
    _emIntlk();
END_FOR
AssertFalse(Condition := _hIA.ExtendOut,
    Message := 'interlocked child must not energize its output (§7)');
_d := _emIntlk.GetFaultSummary();
AssertEquals_DWORD(Expected := TO_DWORD(E_Reason.INTERLOCK_DROPPED),
    Actual := TO_DWORD(_d.ReasonCode),
    Message := 'EM surfaces the interlock reason (§7.2)');
AssertEquals_STRING(Expected := 'ClampIntlk.CylA', Actual := _d.SourcePath,
    Message := 'interlock names the blocked child, not the EM (§6.9)');
// §6.1 HELD rolls up like a fault does, but as information: the EM explains WHICH
// child waits on WHICH condition without entering ERROR or blocking a restart.
AssertTrue(Condition := _emIntlk.Held, Message := 'EM adopts the held child (§8.2)');
AssertFalse(Condition := _emIntlk.Error, Message := 'a held child does not fault the EM');
AssertFalse(Condition := _emIntlk.CylB.Error,
    Message := 'the partner keeps its command instead of being aborted');
// Restoring the condition resumes the join with no operator action.
_emIntlk.CylA.SetAreaSafe(Ok := TRUE, DescriptionKey := '');
FOR _i := 1 TO 6 DO
    _simIntlkA(); _simIntlkB(); _emIntlk();
END_FOR
AssertFalse(Condition := _emIntlk.Held, Message := 'hold clears itself when the child resumes');
AssertTrue(Condition := _emIntlk.OutCmd.Confirmed,
    Message := 'the suspended clamp completes after the interlock returns');
_emIntlk.Execute := FALSE;
_emIntlk();
TEST_FINISHED();
END_METHOD

// §5.7 T5 for the composite tier: a stored ClampEM ParCfg whose SchemaVersion is
// not the expected one must migrate-or-fault with RECIPE_INVALID and never
// mis-run with the wrong parameters (§3.8).
METHOD T5_recipe_schema_mismatch_faults
TEST('T5_recipe_schema_mismatch_faults');
// Setup resolves the recipe, so the fault is raised during construction.
_emBad.Setup(Name := 'ClampBad', HalA := _hBA, HalB := _hBB, Recipe := _prBad);
_emBad();                                    // map ErrorID
AssertTrue(Condition := _emBad.FaultActive,
    Message := 'migrate-or-fault on schema mismatch (§3.8)');
AssertEquals_DWORD(Expected := TO_DWORD(E_Reason.RECIPE_INVALID),
    Actual := _emBad.ErrorID,
    Message := 'RECIPE_INVALID on SchemaVersion mismatch (§3.8)');
// Never mis-runs: a command must not drive an output while the recipe is invalid.
_emBad.Command := E_ClampCommand.CLAMP;
_emBad.Execute := TRUE;
_emBad();
AssertFalse(Condition := _hBA.ExtendOut,
    Message := 'invalid recipe must not mis-run the actuator (§3.8)');
_emBad.Execute := FALSE;
_emBad();
TEST_FINISHED();
END_METHOD

END_FUNCTION_BLOCK

// ---- Fraktal_Tests/FB_ProbeClampCycle.TcPOU
// §6.8 continuous clamp -> unclamp cycle for FB_ProbeClampRoot. Each command
// step names the clamp in Awaits, so a stall or fault is explained by the base
// walk (§6.9) with nothing written here.
FUNCTION_BLOCK FB_ProbeClampCycle EXTENDS FB_SequenceBase
VAR
    {attribute 'OPC.UA.DA' := '0'}
    _clamp : REFERENCE TO FB_ClampEM;
END_VAR

;

METHOD Setup : BOOL
VAR_INPUT
    Host : I_SequenceHost;
END_VAR
VAR_IN_OUT
    Clamp : FB_ClampEM;
END_VAR
_clamp REF= Clamp;
Setup := M_Attach(Host := Host) AND __ISVALIDREF(_clamp);
END_METHOD

METHOD M_Run
CASE _step OF
    0:
        M_Step(StepNo := 0, StepName := 'project.test.clampCycleStart', Awaits := 0,
            AwaitingLabel := '', TimeClass := E_TimeClass.WORK, ExpectedTime := T#0S);
        _retVal := E_StepResult.ADVANCE;
        M_Advance(OnAdvance := 100);
    100:
        M_Step(StepNo := 100, StepName := 'project.test.clamp', Awaits := _clamp,
            AwaitingLabel := 'Clamp.CLAMP', TimeClass := E_TimeClass.WORK, ExpectedTime := T#0S);
        IF M_TryIssue(Steppable := TRUE) THEN
            _clamp.Abort := FALSE;
            _clamp.Command := E_ClampCommand.CLAMP;
            _clamp.Execute := TRUE;
        END_IF
        IF _clamp.Done THEN
            _clamp.Execute := FALSE;
            _retVal := E_StepResult.ADVANCE;
        END_IF
        M_Advance(OnAdvance := 200);
    200:
        M_Step(StepNo := 200, StepName := 'project.test.unclamp', Awaits := _clamp,
            AwaitingLabel := 'Clamp.UNCLAMP', TimeClass := E_TimeClass.WORK, ExpectedTime := T#0S);
        IF M_TryIssue(Steppable := TRUE) THEN
            _clamp.Abort := FALSE;
            _clamp.Command := E_ClampCommand.UNCLAMP;
            _clamp.Execute := TRUE;
        END_IF
        IF _clamp.Done THEN
            _clamp.Execute := FALSE;
            _retVal := E_StepResult.ADVANCE;
        END_IF
        M_Advance(OnAdvance := 999);
    999:
        M_Step(StepNo := 999, StepName := 'project.test.clampCycleComplete', Awaits := 0,
            AwaitingLabel := '', TimeClass := E_TimeClass.WORK, ExpectedTime := T#0S);
        IF M_EndOfCycle() THEN
            _retVal := E_StepResult.ADVANCE;   // no stop requested: next cycle
        END_IF
        M_Advance(OnAdvance := 100);
ELSE
    M_Fault(Reason := E_Reason.STEP_STALLED, DescriptionKey := 'std.error.undefinedStep');
END_CASE
END_METHOD

END_FUNCTION_BLOCK

// ---- Fraktal_Tests/FB_ProbeClampRoot.TcPOU
// §5.7 Unit-tier probe: a root over the library's clamp EM, the shape a project
// Unit takes - wiring only, every step in its chain (§6.8). It replaces the
// library's former FB_ClampStationUnit, a concrete application Unit a reusable
// library must not ship (§6.7); the Unit-tier rows it carried are proven here.
FUNCTION_BLOCK FB_ProbeClampRoot EXTENDS FB_UnitBase
VAR_OUTPUT
    Clamp : FB_ClampEM;
END_VAR
VAR
    Chain : FB_ProbeClampCycle;
END_VAR

Cyclic();

METHOD Setup : BOOL
VAR_INPUT
    Name : STRING(80);
    HalA : REFERENCE TO ST_CylinderHal;
    HalB : REFERENCE TO ST_CylinderHal;
    Recipe : I_RecipeProvider;
END_VAR
_M_SetName(Name);
Setup := Clamp.Setup(Name := CONCAT(Name, '.Clamp'), HalA := HalA, HalB := HalB, Recipe := Recipe)
    AND _M_Register(Child := Clamp)
    AND Chain.Setup(Host := THIS^, Clamp := Clamp);
END_METHOD

METHOD PROTECTED _M_Dispatch
Chain.M_Run();
END_METHOD

END_FUNCTION_BLOCK

// ---- Fraktal_Tests/FB_UnitTier_Tests.TcPOU
// §5.7 suite for the UNIT tier. Rows T1/T4 and the T2/T6/T10 *mechanisms* are
// proven once in the framework base suites (FB_Base_Tests, FB_Unit_Tests,
// FB_Release_Tests) and are NOT re-tested here (§5.7: "types shall not re-test
// inherited rows"). What the Unit tier owes with its OWN modes/paths/actions:
//   T6  cross-tier rollup reaches the ROOT, naming the deepest child
//   T8  mode lifecycle: an unsupported mode is rejected gracefully, no state change
//   T9  stall walk: a stalled step names the awaited module or first FALSE condition
//   T10 gate/report equivalence for THIS unit's actions
// The root is FB_ProbeClampRoot: a project-shaped Unit over the library clamp EM.
FUNCTION_BLOCK FB_UnitTier_Tests EXTENDS TcUnit.FB_TestSuite
VAR
    _station : FB_ProbeClampRoot;
    _halA, _halB : ST_CylinderHal;
    _simA, _simB : FB_CylinderSim;
    _recipe : FB_LocalRecipeProvider;
    _cylinderCfg : ST_CylinderParCfg;
    _clampCfg : ST_ClampParCfg;
    _wired : BOOL;

    // T6/T9 — a second station whose CylB never reaches position (deterministic
    // timeout), so the root can be asked what it is waiting on / what failed.
    _stall : FB_ProbeClampRoot;
    _sHalA, _sHalB : ST_CylinderHal;
    _sSimA : FB_CylinderSim;
    _stallRecipe : FB_LocalRecipeProvider;
    _stallCylCfg : ST_CylinderParCfg;
    _stallClampCfg : ST_ClampParCfg;

    _d : ST_Diagnostic;
    _r : ST_ReleaseReport;
    _ok : BOOL;
    _modeBefore : E_Mode;
    _i : INT;
END_VAR

IF NOT _wired THEN
    _recipe.Register(ModelCode := '', RecipeKey := 'CylinderCM', pData := ADR(_cylinderCfg), Size := SIZEOF(_cylinderCfg));
    _recipe.Register(ModelCode := '', RecipeKey := 'ClampEM', pData := ADR(_clampCfg), Size := SIZEOF(_clampCfg));
    _station.Setup(Name := 'Test.Station', HalA := _halA, HalB := _halB, Recipe := _recipe);
    _simA.Setup(HalRef := _halA, TravelTime := T#0S);
    _simB.Setup(HalRef := _halB, TravelTime := T#0S);
    // Stall/rollup fixture: CylB has no sim plant and a zero move timeout, so the
    // clamp cannot complete and the root must explain why.
    _stallCylCfg.MoveTimeout := T#0S;
    _stallClampCfg.SettleTime := T#0S;
    _stallRecipe.Register(ModelCode := '', RecipeKey := 'CylinderCM', pData := ADR(_stallCylCfg), Size := SIZEOF(_stallCylCfg));
    _stallRecipe.Register(ModelCode := '', RecipeKey := 'ClampEM', pData := ADR(_stallClampCfg), Size := SIZEOF(_stallClampCfg));
    _stall.Setup(Name := 'Stall.Station', HalA := _sHalA, HalB := _sHalB, Recipe := _stallRecipe);
    _sSimA.Setup(HalRef := _sHalA, TravelTime := T#0S);
    _wired := TRUE;
END_IF
Root_is_a_real_unit();
T8_unsupported_mode_is_rejected_gracefully();
T10_start_gate_matches_release_report();
T6_T9_root_rollup_names_deepest_child();

METHOD Root_is_a_real_unit
TEST('Root_is_a_real_unit');
_station();
AssertEquals_DINT(Expected := TO_DINT(E_ModuleType.UNIT),
    Actual := TO_DINT(_station.Status.ModuleType),
    Message := 'demo root publishes Unit identity');
AssertEquals_DINT(Expected := TO_DINT(E_ModuleType.EQUIPMENT_MODULE),
    Actual := TO_DINT(_station.Clamp.Status.ModuleType),
    Message := 'Clamp remains an Equipment Module child');
TEST_FINISHED();
END_METHOD

// §5.7 T10 — gate/report equivalence for THIS unit: Start accepts exactly when
// ReleaseReportStart says Released. Asserting both directions on the same object
// is what proves the report is the authoritative predicate rather than a
// separately-maintained description that can drift from the gate (§7.8).
METHOD T10_start_gate_matches_release_report
TEST('T10_start_gate_matches_release_report');
_station();
_ok := _station.ReleaseReportStart(Report := _r);
// Whatever the current release state is, the gate must agree with it.
AssertEquals_BOOL(Expected := _r.Released, Actual := _ok,
    Message := 'report return value matches the record (7.8)');
IF _r.Released THEN
    AssertTrue(Condition := _station.Start(),
        Message := 'Start accepts exactly when the report is Released (7.8)');
    _station();
    _station.Stop();
    _station();
ELSE
    AssertFalse(Condition := _station.Start(),
        Message := 'Start refuses exactly when the report is not Released (7.8)');
    AssertTrue(Condition := _r.Count > 0,
        Message := 'a refusal must list at least one concrete reason (7.8)');
END_IF
TEST_FINISHED();
END_METHOD

// §5.7 T6 + T9 at the ROOT. T6: the first-out must be adopted VERBATIM up two
// tiers (Cyl -> Clamp EM -> Unit), naming the deepest failing child rather than
// the nearest parent — that two-hop walk is what the Unit tier adds over the EM's
// single hop. T9: the root's diagnostic must name the module it was waiting on,
// so a stalled station is diagnosable without opening XAE (§6.9(b)).
METHOD T6_T9_root_rollup_names_deepest_child
TEST('T6_T9_root_rollup_names_deepest_child');
// CylB has no sim plant and MoveTimeout T#0S, so the clamp cannot complete.
_ok := _stall.Start();
FOR _i := 1 TO 12 DO
    _stall();
    _sSimA();                                // CylA completes; CylB never arrives
END_FOR
_d := _stall.GetFaultSummary();
AssertEquals_STRING(Expected := 'Stall.Station.Clamp.CylB', Actual := _d.SourcePath,
    Message := 'root adopts the deepest child path verbatim across two tiers (8.2)');
AssertEquals_DWORD(Expected := TO_DWORD(PL_ModuleReasons.CYL_NOT_EXTENDED),
    Actual := TO_DWORD(_d.ReasonCode),
    Message := 'reason code is the childs, not a generic parent code (8.2)');
AssertTrue(Condition := _d.SourcePath <> 'Stall.Station',
    Message := 'the root must not name itself as the source (6.9)');
_stall.Stop();
_stall();
TEST_FINISHED();
END_METHOD

// §5.7 T8 — mode lifecycle for THIS unit's mode set. FB_ProbeClampRoot does not
// override _M_Supports, so its set is the baseline AUTO + MANUAL: requesting
// CALIBRATION must be refused *gracefully* — SetMode returns FALSE, the active
// mode is unchanged, and the unit does not fault (a rejected request is not an
// error, §3.7).
METHOD T8_unsupported_mode_is_rejected_gracefully
TEST('T8_unsupported_mode_is_rejected_gracefully');
_station();
_modeBefore := _station.ModeActive;
_ok := _station.SetMode(Mode := E_Mode.CALIBRATION);
AssertFalse(Condition := _ok,
    Message := 'unsupported mode returns FALSE, not a fault (3.7)');
_station();
AssertEquals_DINT(Expected := TO_DINT(_modeBefore),
    Actual := TO_DINT(_station.ModeActive),
    Message := 'rejected request leaves the active mode unchanged (3.7)');
AssertFalse(Condition := _station.Error,
    Message := 'graceful rejection must not raise a module error (3.7)');
// A supported mode from the same set is still accepted afterwards.
AssertTrue(Condition := _station.SetMode(Mode := E_Mode.MANUAL),
    Message := 'supported mode still accepted after a rejection');
FOR _i := 1 TO 4 DO
    _station();
END_FOR
AssertEquals_DINT(Expected := TO_DINT(E_Mode.MANUAL),
    Actual := TO_DINT(_station.ModeActive),
    Message := 'supported mode commits (3.4)');
_station.SetMode(Mode := E_Mode.AUTO);
FOR _i := 1 TO 4 DO
    _station();
END_FOR
TEST_FINISHED();
END_METHOD

END_FUNCTION_BLOCK

// ---- Fraktal_Tests/FB_Connector_Tests.TcPOU
// FB_DeviceConnectorBase suite — row T7 (link supervision) proven once (5.7)
FUNCTION_BLOCK FB_Connector_Tests EXTENDS TcUnit.FB_TestSuite
VAR
    _c1, _c2 : FB_ProbeConnector;
    _w : BOOL;
    _d : ST_Diagnostic;
END_VAR

Heartbeat_links_and_protocol_fail_drops();
Silent_link_confirms_LINK_TIMEOUT();
Module_contract_is_neutral();

METHOD Heartbeat_links_and_protocol_fail_drops
TEST('Heartbeat_links_and_protocol_fail_drops');
IF NOT _w THEN
    _c1.Setup('Test.Link1');
    _c1.HbPeriod := T#0S;
    _c1.LinkTimeout := T#1H;                 // loss confirm never fires in this test
    _c2.Setup('Test.Link2');
    _c2.HbPeriod := T#1H;                    // heartbeat never due
    _c2.LinkTimeout := T#0S;                 // loss confirms immediately
    _w := TRUE;
END_IF
AssertTrue(Condition := _c1.Connect(), Message := 'session opens');
_c1();                                       // hb due -> start
_c1();                                       // poll OK -> Linked
AssertTrue(Condition := _c1.Linked, Message := 'healthy heartbeat links (3.15.2)');
_c1.SimHb := E_HbResult.FAIL;
_c1();                                       // hb start
_c1();                                       // poll FAIL -> protocol error, session dropped
AssertFalse(Condition := _c1.Linked, Message := 'protocol failure drops the link');
_d := _c1.LinkReason;
AssertEquals_DWORD(Expected := TO_DWORD(E_Reason.DEVICE_PROTOCOL_ERROR),
                   Actual   := TO_DWORD(_d.ReasonCode),
                   Message  := 'first-out names the protocol error');
AssertEquals_STRING(Expected := 'Test.Link1', Actual := _d.SourcePath,
                    Message := 'link reason names the connector path (6.9)');
AssertTrue(Condition := _c1.FaultActive, Message := 'connector reports FaultActive for rollup');
TEST_FINISHED();
END_METHOD

METHOD Silent_link_confirms_LINK_TIMEOUT
TEST('Silent_link_confirms_LINK_TIMEOUT');
AssertTrue(Condition := _c2.Connect(), Message := 'session opens');
_c2();                                       // no beat; loss confirm (T#0S) -> LINK_TIMEOUT
AssertFalse(Condition := _c2.Linked, Message := 'silent device drops the link');
_d := _c2.LinkReason;
AssertEquals_DWORD(Expected := TO_DWORD(E_Reason.LINK_TIMEOUT),
                   Actual   := TO_DWORD(_d.ReasonCode),
                   Message  := 'LINK_TIMEOUT confirmed after LinkTimeout (3.15.2)');
TEST_FINISHED();
END_METHOD

METHOD Module_contract_is_neutral
TEST('Module_contract_is_neutral');
AssertTrue(Condition := _c1.M_ReleaseCommand(),
           Message := 'connector accepts generic command release without changing link ownership');
AssertFalse(Condition := _c1.HoldActive,
            Message := 'fronting Control Module, not connector, owns HELD state');
TEST_FINISHED();
END_METHOD

END_FUNCTION_BLOCK

// ---- Fraktal_Tests/FB_CylinderCM_Tests.TcPOU
// Annex H suite for the cylinder TYPE: T2/T3/T5 with ITS reasons + functional
// completion against the sim plant model (T1/T4 inherited — not repeated, §5.7).
FUNCTION_BLOCK FB_CylinderCM_Tests EXTENDS TcUnit.FB_TestSuite
VAR
    _cm1, _cm2, _cm3, _cm4, _cm5, _cm6 : FB_CylinderCM;
    _h1, _h2, _h3, _h4, _h5, _h6 : ST_CylinderHal;
    _sim1 : FB_CylinderSim;
    _prOk, _prFast, _prBad : FB_LocalRecipeProvider;
    _bOk, _bFast, _bBad : ST_CylinderParCfg;
    _prModels : FB_LocalRecipeProvider;
    _modelA, _modelB, _loaded : ST_CylinderParCfg;
    _d : ST_Diagnostic;
    _release : ST_ReleaseReport;
    _io6 : ST_CylinderIoIdentity;
    _w : BOOL;
END_VAR

IF NOT _w THEN
    _bFast.MoveTimeout := T#0S;              // deterministic timeout in one scan
    _bBad.SchemaVersion := 2;                // stored schema != expected (=1)
    _prOk.Register(ModelCode := '', RecipeKey := 'CylinderCM', pData := ADR(_bOk), Size := SIZEOF(_bOk));
    _prFast.Register(ModelCode := '', RecipeKey := 'CylinderCM', pData := ADR(_bFast), Size := SIZEOF(_bFast));
    _prBad.Register(ModelCode := '', RecipeKey := 'CylinderCM', pData := ADR(_bBad), Size := SIZEOF(_bBad));
    _modelA.MoveTimeout := T#1S;
    _modelB.MoveTimeout := T#2S;
    _prModels.Register(ModelCode := 'A', RecipeKey := 'CylinderCM', pData := ADR(_modelA), Size := SIZEOF(_modelA));
    _prModels.Register(ModelCode := 'B', RecipeKey := 'CylinderCM', pData := ADR(_modelB), Size := SIZEOF(_modelB));
    _cm1.Setup(Name := 'Test.Cyl1', HalRef := _h1, Recipe := _prOk);
    _sim1.Setup(HalRef := _h1, TravelTime := T#0S);
    _cm2.Setup(Name := 'Test.Cyl2', HalRef := _h2, Recipe := _prFast);
    _cm3.Setup(Name := 'Test.Cyl3', HalRef := _h3, Recipe := _prOk);
    _cm5.Setup(Name := 'Test.Cyl5', HalRef := _h5, Recipe := _prOk);
    _cm6.Setup(Name := 'Test.Cyl6', HalRef := _h6, Recipe := _prFast);
    _io6.ExtendedSensor.Tag := '_101B202A';
    _io6.ExtendedSensor.Address := 'EL1809 Ch5';
    _io6.RetractedSensor.Tag := '_101B202B';
    _io6.RetractedSensor.Address := 'EL1809 Ch6';
    _io6.ExtendOutput.Tag := '_101K202A';
    _io6.RetractOutput.Tag := '_101K202B';
    _io6.ExtendedTimeoutKey := 'project.error.pressDownSensorTimeout';
    _io6.RetractedTimeoutKey := 'project.error.pressUpSensorTimeout';
    _io6.BothSensorsKey := 'project.error.pressPositionSensorsConflict';
    _cm6.ConfigureIoIdentity(Identity := _io6);
    _w := TRUE;
END_IF
Extend_completes_against_sim();
T2_first_out_reason_and_path();
T3_interlock_withholds_output();
T5_recipe_schema_mismatch_faults();
Recipe_lookup_uses_model_and_key();
Directional_interlock_covers_typed_command();
Timeout_identifies_sensor_tag();

METHOD Extend_completes_against_sim
TEST('Extend_completes_against_sim');
_cm1.Command := E_CylinderCommand.EXTEND;
_cm1.Execute := TRUE;
_cm1();                                      // edge -> step 10 drives ExtendOut
_cm1();                                      // step 20 awaiting fb
_sim1();                                     // plant: sensor made (travel T#0S)
_cm1();                                      // sees fb -> Done
AssertTrue(Condition := _cm1.Done, Message := 'handshake completes on feedback (6.1)');
AssertTrue(Condition := _cm1.Timing.Rows[1].Count = 1,
           Message := 'command timing row captured (8.11.4a)');
_cm1.Execute := FALSE;
_cm1();
TEST_FINISHED();
END_METHOD

METHOD Directional_interlock_covers_typed_command
TEST('Directional_interlock_covers_typed_command');
_cm5.SetDirectionalPermits(ExtendOk := FALSE, RetractOk := TRUE,
    ExtendDescriptionKey := 'project.interlock.testExtendBlocked',
    RetractDescriptionKey := 'project.interlock.testRetractAllowed');
_cm5.AppendDirectionalRelease(Value := TO_DINT(E_CylinderCommand.EXTEND), Report := _release);
AssertTrue(Condition := _release.Count = 1,
    Message := 'manual release query reports the selected blocked direction');
AssertEquals_STRING(Expected := 'project.interlock.testExtendBlocked',
    Actual := _release.Reasons[1].Description, Message := 'release query and dispatch share one key');
AssertEquals_STRING(Expected := 'Test.Cyl5', Actual := _release.Reasons[1].SourcePath,
    Message := 'directional release preserves the child module path');
_cm5.Command := E_CylinderCommand.EXTEND;
_cm5.Execute := TRUE;
_cm5();
AssertFalse(Condition := _h5.ExtendOut,
    Message := 'direction-specific collision interlock withholds output');
AssertEquals_DWORD(Expected := TO_DWORD(E_Reason.INTERLOCK_DROPPED),
    Actual := _cm5.ErrorID, Message := 'direction interlock uses common reason');
_d := _cm5.GetFaultSummary();
AssertEquals_STRING(Expected := 'project.interlock.testExtendBlocked',
    Actual := _d.Description, Message := 'selected direction publishes its key');
TEST_FINISHED();
END_METHOD

METHOD T2_first_out_reason_and_path
TEST('T2_first_out_reason_and_path');
_cm2.Command := E_CylinderCommand.EXTEND;
_cm2.Execute := TRUE;
_cm2();                                      // step 10
_cm2();                                      // step 20: MoveTimeout T#0S -> fault
AssertTrue(Condition := _cm2.Error, Message := 'Error after MoveTimeout');
AssertEquals_DWORD(Expected := TO_DWORD(PL_ModuleReasons.CYL_NOT_EXTENDED),
                   Actual   := _cm2.ErrorID,
                   Message  := 'first-out is the type band code 10101 (8.8)');
_d := _cm2.GetFaultSummary();
AssertEquals_STRING(Expected := 'Test.Cyl2', Actual := _d.SourcePath,
                    Message := 'reason names the source path (6.9)');
TEST_FINISHED();
END_METHOD

METHOD T3_interlock_withholds_output
TEST('T3_interlock_withholds_output');
_cm3.SetAreaSafe(Ok := FALSE, DescriptionKey := '');   // the real §7.2 path
_cm3.Command := E_CylinderCommand.EXTEND;
_cm3.Execute := TRUE;
_cm3();
AssertFalse(Condition := _h3.ExtendOut,
            Message := 'output must not energize while interlocked (7)');
AssertEquals_DWORD(Expected := TO_DWORD(E_Reason.INTERLOCK_DROPPED),
                   Actual   := _cm3.ErrorID,
                   Message  := 'interlock reason expected (7.2)');
_d := _cm3.GetFaultSummary();
AssertEquals_STRING(Expected := 'Test.Cyl3', Actual := _d.SourcePath,
                    Message := 'owner sets the source path (7.2)');
// 6.1 HELD — an interlock lost during a command suspends the command, it does not
// fail it: no ERROR to reset, no MANUAL_RESET alarm, and the reason is LOW.
AssertTrue(Condition := _cm3.Held, Message := 'interlocked command is HELD (6.1)');
AssertFalse(Condition := _cm3.Error, Message := 'a lost interlock is not a fault');
AssertTrue(Condition := _cm3.Busy, Message := 'held command stays BUSY so its owner keeps awaiting it');
AssertEquals_DINT(Expected := TO_DINT(E_Severity.LOW), Actual := TO_DINT(_d.Severity),
                  Message := 'a declared wait is LOW, not a downtime event (8.1/8.4)');
// ...and restoring the condition resumes it with no operator action at all.
_cm3.SetAreaSafe(Ok := TRUE, DescriptionKey := '');
_cm3();
AssertFalse(Condition := _cm3.Held, Message := 'hold clears itself when the condition returns');
AssertTrue(Condition := _h3.ExtendOut, Message := 'resume re-energizes the direction output');
AssertEquals_DWORD(Expected := 0, Actual := _cm3.ErrorID,
                   Message := 'the resumed command carries no lingering reason');
_cm3.Execute := FALSE;
_cm3();
TEST_FINISHED();
END_METHOD

METHOD T5_recipe_schema_mismatch_faults
TEST('T5_recipe_schema_mismatch_faults');
_cm4.Setup(Name := 'Test.Cyl4', HalRef := _h4, Recipe := _prBad);   // stored v2 vs expected v1
_cm4();                                      // map ErrorID
AssertTrue(Condition := _cm4.FaultActive, Message := 'migrate-or-fault (3.8)');
AssertEquals_DWORD(Expected := TO_DWORD(E_Reason.RECIPE_INVALID),
                   Actual   := _cm4.ErrorID,
                   Message  := 'RECIPE_INVALID on SchemaVersion mismatch (3.8)');
TEST_FINISHED();
END_METHOD

METHOD Recipe_lookup_uses_model_and_key
TEST('Recipe_lookup_uses_model_and_key');
AssertTrue(Condition := _prModels.Load(ModelCode := 'B', RecipeKey := 'CylinderCM',
    pParCfg := ADR(_loaded), Size := SIZEOF(_loaded)),
    Message := 'model-specific record found');
AssertTrue(Condition := _loaded.MoveTimeout = T#2S,
    Message := 'same recipe key resolves by ModelCode');
TEST_FINISHED();
END_METHOD

METHOD Timeout_identifies_sensor_tag
TEST('Timeout_identifies_sensor_tag');
_cm6.Command := E_CylinderCommand.EXTEND;
_cm6.Execute := TRUE;
_cm6();
_cm6();
_d := _cm6.GetFaultSummary();
AssertEquals_STRING(Expected := '_101B202A', Actual := _d.IoTag,
    Message := 'timeout carries exact schematic sensor tag');
AssertEquals_STRING(Expected := 'EL1809 Ch5', Actual := _d.IoAddress,
    Message := 'timeout carries terminal channel locator');
AssertEquals_STRING(Expected := 'project.error.pressDownSensorTimeout',
    Actual := _d.Description, Message := 'timeout uses project-localizable sensor message');
TEST_FINISHED();
END_METHOD

END_FUNCTION_BLOCK

// ---- Fraktal_Tests/FB_Decision_Tests.TcPOU
// Core §6.11: one active request, safe resolution, timeout/default and audit.
FUNCTION_BLOCK FB_Decision_Tests EXTENDS TcUnit.FB_TestSuite
VAR
    _operator : FB_ProbeUnit;
    _overlap  : FB_ProbeUnit;
    _timeout  : FB_ProbeUnit;
    _invalid  : FB_ProbeUnit;
    _operatorReq : ST_DecisionRequest;
    _overlapReq  : ST_DecisionRequest;
    _otherReq    : ST_DecisionRequest;
    _timeoutReq  : ST_DecisionRequest;
    _invalidReq  : ST_DecisionRequest;
    _report : ST_ReleaseReport;
    _wOperator, _wOverlap, _wTimeout, _wInvalid : BOOL;
    _ringHead : INT;
END_VAR

Operator_choice_is_validated_consumed_and_logged();
Repeated_request_is_idempotent_and_overlap_rejects();
Timeout_uses_the_validated_safe_default();
Invalid_timeout_default_faults_without_publication();

METHOD Operator_choice_is_validated_consumed_and_logged
VAR
    answer : INT;
END_VAR
TEST('Operator_choice_is_validated_consumed_and_logged');
IF NOT _wOperator THEN
    _operator.Setup(Name := 'Test.DecisionOperator');
    AssertTrue(Condition := _operator.Start(), Message := 'Unit starts');
    _operator();
    _operatorReq.Prompt := 'project.decision.operator';
    _operatorReq.Options[1] := 'project.option.retry';
    _operatorReq.Options[2] := 'project.option.continue';
    _operatorReq.Default := 1;
    _operatorReq.Timeout := T#5S;
    AssertTrue(Condition := _operator.M_TestAskDecision(Req := _operatorReq),
        Message := 'valid request is published');
    AssertTrue(Condition := _operator.SubmitDecision(Option := 2, Report := _report),
        Message := 'active published option is accepted through the authoritative entry');
    _operator();
    answer := _operator.M_TestTakeDecision();
    AssertEquals_INT(Expected := 2, Actual := answer,
        Message := 'answer is consumed exactly once');
    AssertEquals_STRING(Expected := '', Actual := _operator.Decision.Prompt,
        Message := 'consumption clears the complete public slot');
    AssertEquals_STRING(Expected := 'std.audit.decisionOperatorResolved option=2',
        Actual := _operator.AlarmLog.Ring[_operator.AlarmLog.RingHead].Description,
        Message := 'operator resolution is a domain audit event');
    _wOperator := TRUE;
END_IF
TEST_FINISHED();
END_METHOD

METHOD Repeated_request_is_idempotent_and_overlap_rejects
TEST('Repeated_request_is_idempotent_and_overlap_rejects');
IF NOT _wOverlap THEN
    _overlap.Setup(Name := 'Test.DecisionOverlap');
    AssertTrue(Condition := _overlap.Start(), Message := 'Unit starts');
    _overlap();
    _overlapReq.Prompt := 'project.decision.first';
    _overlapReq.Options[1] := 'project.option.ok';
    _overlapReq.Timeout := T#0S;
    _otherReq.Prompt := 'project.decision.second';
    _otherReq.Options[1] := 'project.option.cancel';
    _otherReq.Timeout := T#0S;
    AssertTrue(Condition := _overlap.M_TestAskDecision(Req := _overlapReq),
        Message := 'first request owns the slot');
    _ringHead := _overlap.AlarmLog.RingHead;
    AssertTrue(Condition := _overlap.M_TestAskDecision(Req := _overlapReq),
        Message := 'same request is idempotent');
    AssertEquals_INT(Expected := _ringHead, Actual := _overlap.AlarmLog.RingHead,
        Message := 'idempotent presentation does not duplicate request audit');
    AssertFalse(Condition := _overlap.M_TestAskDecision(Req := _otherReq),
        Message := 'different request cannot overwrite the active slot');
    AssertEquals_STRING(Expected := 'project.decision.first', Actual := _overlap.Decision.Prompt,
        Message := 'first producer retains ownership');
    AssertEquals_STRING(Expected := 'std.audit.decisionOverlapRejected',
        Actual := _overlap.AlarmLog.Ring[_overlap.AlarmLog.RingHead].Description,
        Message := 'overlap is rejected and logged');
    _ringHead := _overlap.AlarmLog.RingHead;
    AssertFalse(Condition := _overlap.M_TestAskDecision(Req := _otherReq),
        Message := 'repeated conflict remains rejected');
    AssertEquals_INT(Expected := _ringHead, Actual := _overlap.AlarmLog.RingHead,
        Message := 'one repeated producer cannot flood the bounded event ring');
    _overlap.M_TestClearDecision();
    _wOverlap := TRUE;
END_IF
TEST_FINISHED();
END_METHOD

METHOD Timeout_uses_the_validated_safe_default
VAR
    answer : INT;
END_VAR
TEST('Timeout_uses_the_validated_safe_default');
IF NOT _wTimeout THEN
    _timeout.Setup(Name := 'Test.DecisionTimeout');
    AssertTrue(Condition := _timeout.Start(), Message := 'Unit starts');
    _timeout();
    _timeoutReq.Prompt := 'project.decision.timeout';
    _timeoutReq.Options[1] := 'project.option.safeStop';
    _timeoutReq.Options[2] := 'project.option.continue';
    _timeoutReq.Default := 1;
    _timeoutReq.Timeout := T#1MS;
    AssertTrue(Condition := _timeout.M_TestAskDecision(Req := _timeoutReq),
        Message := 'timed request is published');
    _wTimeout := TRUE;
ELSE
    _timeout();
    IF _timeout.DecisionAnswer > 0 THEN
        answer := _timeout.M_TestTakeDecision();
        AssertEquals_INT(Expected := 1, Actual := answer,
            Message := 'timeout resolves to the validated safe default');
        AssertEquals_STRING(Expected := 'std.audit.decisionTimeoutResolved option=1',
            Actual := _timeout.AlarmLog.Ring[_timeout.AlarmLog.RingHead].Description,
            Message := 'timeout origin is explicit in the audit');
        TEST_FINISHED();
    END_IF
END_IF
END_METHOD

METHOD Invalid_timeout_default_faults_without_publication
TEST('Invalid_timeout_default_faults_without_publication');
IF NOT _wInvalid THEN
    _invalid.Setup(Name := 'Test.DecisionInvalid');
    AssertTrue(Condition := _invalid.Start(), Message := 'Unit starts');
    _invalid();
    _invalidReq.Prompt := 'project.decision.invalid';
    _invalidReq.Options[1] := 'project.option.safeStop';
    _invalidReq.Default := 2;
    _invalidReq.Timeout := T#1S;
    AssertFalse(Condition := _invalid.M_TestAskDecision(Req := _invalidReq),
        Message := 'missing default option is rejected');
    _invalid();
    AssertTrue(Condition := _invalid.Error,
        Message := 'invalid application request faults on the lifecycle output mapping');
    AssertEquals_STRING(Expected := '', Actual := _invalid.Decision.Prompt,
        Message := 'invalid request is never published');
    _wInvalid := TRUE;
END_IF
TEST_FINISHED();
END_METHOD

END_FUNCTION_BLOCK

// ---- Fraktal_Tests/FB_Hmi_Tests.TcPOU
// §3.10(a') under test: the data mirror IS the HMI contract — proven once.
FUNCTION_BLOCK FB_Hmi_Tests EXTENDS TcUnit.FB_TestSuite
VAR
    _p : FB_ProbeCM;
    _u : FB_ProbeUnit;
    _invalidNokUnit : FB_ProbeUnit;
    _mailboxUnit : FB_ProbeUnit;
    _mailboxInit : BOOL;
    _policyUnit : FB_ProbeUnit;
    _policyInit : BOOL;
    _policyProvider : FB_LocalAccessProvider;
    _w : BOOL;
END_VAR

Status_mirror_carries_name_state_and_diag();
Unit_publishes_counters_and_history();
Nameplate_roundtrip();
Mailbox_commits_once_and_acknowledges();
Mailbox_policy_is_self_gated_and_power_ack_is_authoritative();

METHOD Status_mirror_carries_name_state_and_diag
TEST('Status_mirror_carries_name_state_and_diag');
IF NOT _w THEN
    _p.Setup('Test.Mirror');
    _u.Setup('Test.MirrorUnit');
    _invalidNokUnit.Setup('Test.InvalidNokUnit');
    _w := TRUE;
END_IF
AssertEquals_STRING(Expected := 'Test.Mirror', Actual := _p.Status.Name,
                    Message := 'mirror carries the browse name (3.10a$')');
_p.Execute := TRUE;
_p.SimFault := TRUE;
_p();
AssertEquals_DINT(Expected := TO_DINT(E_ExecState.ERROR),
                  Actual   := TO_DINT(_p.Status.State),
                  Message  := 'mirror state follows ExecState');
AssertEquals_DWORD(Expected := TO_DWORD(E_Reason.TEST_FAULT),
                   Actual   := TO_DWORD(_p.Status.Diagnostic.ReasonCode),
                   Message  := 'live diagnostic published as DATA (6.9a)');
AssertEquals_DINT(Expected := TO_DINT(E_Severity.LOW),
    Actual := TO_DINT(_p.Status.Diagnostic.Severity),
    Message := 'diagnostic uses the generated reason priority at its source');
AssertEquals_DINT(Expected := TO_DINT(E_Category.SYSTEM),
    Actual := TO_DINT(_p.Status.Diagnostic.Category),
    Message := 'diagnostic uses the generated reason category at its source');
AssertTrue(Condition := _p.Status.FaultActive, Message := 'mirror fault flag');
_p.Execute := FALSE;
_p.SimFault := FALSE;
_p();
TEST_FINISHED();
END_METHOD

METHOD Unit_publishes_counters_and_history
TEST('Unit_publishes_counters_and_history');
AssertFalse(Condition := _invalidNokUnit.CountNok(Reason := E_Reason.NONE),
    Message := 'unattributed NOK rejected');
AssertEquals_UDINT(Expected := 0, Actual := _invalidNokUnit.NokCount,
    Message := 'rejected NOK does not alter KPI');
AssertEquals_INT(Expected := 0, Actual := _invalidNokUnit.HostEvents.Count,
    Message := 'rejected NOK does not publish a host event');
_u.CountGood();
_u.CountGood();
AssertTrue(Condition := _u.CountNok(Reason := E_Reason.RESULT_RECORD_REJECTED),
    Message := 'attributed NOK accepted without optional carrier');
AssertEquals_UDINT(Expected := 2, Actual := _u.GoodCount, Message := 'good counter (8.11)');
AssertEquals_UDINT(Expected := 1, Actual := _u.NokCount,  Message := 'nok counter (8.11)');
AssertEquals_DINT(Expected := TO_DINT(E_HostEventKind.NOK),
    Actual := TO_DINT(_u.HostEvents.Ring[_u.HostEvents.RingHead].Kind),
    Message := 'NOK host event emitted without optional carrier (11.6)');
AssertEquals_DWORD(Expected := TO_DWORD(E_Reason.RESULT_RECORD_REJECTED),
    Actual := TO_DWORD(_u.HostEvents.Ring[_u.HostEvents.RingHead].ReasonCode),
    Message := 'NOK host event preserves first-out reason');
// stall pending surfaces on the mirror while no fault is active (6.9/3.10a')
AssertTrue(Condition := _u.Start(), Message := 'start');
_u();
_u();                                        // StallTime T#0S -> pending
AssertEquals_DWORD(Expected := TO_DWORD(E_Reason.STEP_STALLED),
                   Actual   := TO_DWORD(_u.Status.Diagnostic.ReasonCode),
                   Message  := 'pending stall visible on the data mirror');
_u.Stop();
_u.SimA := TRUE;
_u.SimB := TRUE;
_u();
_u();
_u();
TEST_FINISHED();
END_METHOD

// §3.10.1: SetNameplate persists identity; published for the HMI facet card
METHOD Nameplate_roundtrip
VAR
    plate : ST_Nameplate;
END_VAR
TEST('Nameplate_roundtrip');
plate.ManufacturerName := 'ACME';
plate.SerialNumber := 'SN-1';
_p.SetNameplate(Plate := plate);
AssertEquals_STRING(Expected := 'ACME', Actual := _p.Nameplate.ManufacturerName, Message := 'manufacturer persists');
AssertEquals_STRING(Expected := 'SN-1', Actual := _p.Nameplate.SerialNumber, Message := 'serial persists');
TEST_FINISHED();
END_METHOD

// §3.10(a″): arguments are sampled only when Sequence changes; Ack is last.
METHOD Mailbox_commits_once_and_acknowledges
TEST('Mailbox_commits_once_and_acknowledges');
IF NOT _mailboxInit THEN
    _mailboxUnit.Setup('Test.MailboxUnit');
    _mailboxInit := TRUE;
ELSE
    _mailboxInit := _mailboxInit;
END_IF
_mailboxUnit.HmiRequest.Kind := E_HmiRequestKind.SET_MODE;
_mailboxUnit.HmiRequest.IntValue := TO_DINT(E_Mode.MANUAL);
_mailboxUnit.HmiRequest.Sequence := 1;
_mailboxUnit();
AssertEquals_UDINT(Expected := 1, Actual := _mailboxUnit.HmiResponse.AckSequence,
    Message := 'committed sequence acknowledged');
AssertTrue(Condition := _mailboxUnit.HmiResponse.Accepted,
    Message := 'existing gated SetMode path accepted');
AssertEquals_DINT(Expected := TO_DINT(E_Mode.MANUAL),
    Actual := TO_DINT(_mailboxUnit.ModeActivePublished),
    Message := 'property-only mode is published as OPC UA data');

// Change arguments without changing Sequence: the transaction shall not replay.
_mailboxUnit.HmiRequest.IntValue := TO_DINT(E_Mode.AUTO);
_mailboxUnit();
AssertEquals_DINT(Expected := TO_DINT(E_Mode.MANUAL),
    Actual := TO_DINT(_mailboxUnit.ModeActivePublished),
    Message := 'unchanged sequence is ignored');
TEST_FINISHED();
END_METHOD

METHOD Mailbox_policy_is_self_gated_and_power_ack_is_authoritative
TEST('Mailbox_policy_is_self_gated_and_power_ack_is_authoritative');
IF NOT _policyInit THEN
    _policyUnit.Setup('Test.PolicyMailboxUnit');
    // Not under test here: a volatile table, so no previous run's file is a precondition.
    _policyProvider.M_UseKey(Key := '');
    _policyProvider.Register(User := 'admin1', Pin := '4711',
        Level := E_AccessLevel.ADMIN);
    _policyUnit();
    _policyUnit.Access.Setup(Provider := _policyProvider,
        pAlarmLog := ADR(_policyUnit.AlarmLog));
    // Policy is intentionally PERSISTENT. Commission every entry this repeatable
    // fixture observes so a previous successful run cannot become its precondition.
    _policyUnit.Access.ConfigureRequired(Gate := E_GatedAction.ACCESS_POLICY,
        Level := E_AccessLevel.NONE);
    _policyUnit.Access.ConfigureRequired(Gate := E_GatedAction.DATA_WRITE,
        Level := E_AccessLevel.NONE);
    _policyUnit.Access.ConfigureRequired(Gate := E_GatedAction.POWER_CONTROL,
        Level := E_AccessLevel.ADMIN);
    _policyInit := TRUE;
ELSE
    _policyInit := _policyInit;
END_IF

_policyUnit.HmiRequest.Kind := E_HmiRequestKind.CONTROL_ON;
_policyUnit.HmiRequest.Sequence := 1;
_policyUnit();
AssertFalse(Condition := _policyUnit.HmiResponse.Accepted,
    Message := 'control-power acknowledgement reflects PLC authorization');
AssertFalse(Condition := _policyUnit.ReqControlOn,
    Message := 'denied power request never latches');

_policyUnit.HmiRequest.Kind := E_HmiRequestKind.SET_ACCESS_LEVEL;
_policyUnit.HmiRequest.IntValue := TO_DINT(E_GatedAction.ACCESS_POLICY);
_policyUnit.HmiRequest.TextValue := '4';
_policyUnit.HmiRequest.Sequence := 2;
_policyUnit();
AssertFalse(Condition := _policyUnit.HmiResponse.Accepted,
    Message := 'anonymous session cannot raise ACCESS_POLICY above itself');
AssertEquals_DINT(Expected := TO_DINT(E_AccessLevel.NONE),
    Actual := TO_DINT(_policyUnit.Access.Policy.Required[TO_INT(E_GatedAction.ACCESS_POLICY)]),
    Message := 'self-lockout attempt leaves policy open');

_policyUnit.Access.RequestLogin(User := 'admin1', Secret := '4711');
_policyUnit();
_policyUnit.HmiRequest.Sequence := 3;
_policyUnit();
AssertTrue(Condition := _policyUnit.HmiResponse.Accepted,
    Message := 'authenticated admin may raise ACCESS_POLICY to ADMIN');
AssertEquals_DINT(Expected := TO_DINT(E_AccessLevel.ADMIN),
    Actual := TO_DINT(_policyUnit.Access.Policy.Required[TO_INT(E_GatedAction.ACCESS_POLICY)]),
    Message := 'ACCESS_POLICY threshold persisted');

_policyUnit.HmiRequest.IntValue := TO_DINT(E_GatedAction.DATA_WRITE);
_policyUnit.HmiRequest.TextValue := '2';
_policyUnit.Access.RequestLogout();
_policyUnit();
_policyUnit.HmiRequest.Sequence := 4;
_policyUnit();
AssertFalse(Condition := _policyUnit.HmiResponse.Accepted,
    Message := 'policy edits are self-gated after commissioning');
AssertEquals_DINT(Expected := TO_DINT(E_AccessLevel.NONE),
    Actual := TO_DINT(_policyUnit.Access.Policy.Required[TO_INT(E_GatedAction.DATA_WRITE)]),
    Message := 'denied edit leaves target threshold unchanged');
TEST_FINISHED();
END_METHOD

END_FUNCTION_BLOCK

// ---- Fraktal_Tests/FB_HostEvent_Tests.TcPOU
// Core §11.6: fixed event vocabulary, required shape, bounds, and invalid-input rejection.
FUNCTION_BLOCK FB_HostEvent_Tests EXTENDS TcUnit.FB_TestSuite
VAR
    ShapePublisher : FB_HostEventPublisher;
    VocabularyPublisher : FB_HostEventPublisher;
    WrapPublisher : FB_HostEventPublisher;
END_VAR

Rejects_invalid_event();
Publishes_required_shape();
Accepts_fixed_vocabulary();
Ring_is_bounded();

METHOD Rejects_invalid_event
TEST('Rejects_invalid_event');
AssertFalse(Condition := ShapePublisher.Emit(Kind := E_HostEventKind.NONE,
    StationPath := 'U', PartUid := '', Subject := '', Value := '', Verdict := E_Verdict.NONE,
    ReasonCode := E_Reason.NONE), Message := 'NONE is not a host event');
AssertFalse(Condition := ShapePublisher.Emit(Kind := E_HostEventKind.MODE_CHANGED,
    StationPath := '', PartUid := '', Subject := 'Mode', Value := '1', Verdict := E_Verdict.NONE,
    ReasonCode := E_Reason.NONE), Message := 'station path is mandatory');
TEST_FINISHED();
END_METHOD

METHOD Publishes_required_shape
TEST('Publishes_required_shape');
AssertTrue(Condition := ShapePublisher.Emit(Kind := E_HostEventKind.NOK,
    StationPath := 'Root', PartUid := 'P-42', Subject := '', Value := '',
    Verdict := E_Verdict.NOK, ReasonCode := E_Reason.RESULT_RECORD_REJECTED),
    Message := 'valid event accepted');
AssertEquals_UDINT(Expected := 1, Actual := ShapePublisher.Ring[1].Sequence,
    Message := 'monotonic sequence assigned');
AssertEquals_STRING(Expected := 'Root', Actual := ShapePublisher.Ring[1].StationPath,
    Message := 'station browse path carried');
AssertEquals_STRING(Expected := 'P-42', Actual := ShapePublisher.Ring[1].PartUid,
    Message := 'part uid carried when applicable');
AssertEquals_DINT(Expected := TO_DINT(E_Verdict.NOK),
    Actual := TO_DINT(ShapePublisher.Ring[1].Verdict), Message := 'verdict carried');
AssertEquals_DINT(Expected := TO_DINT(E_Reason.RESULT_RECORD_REJECTED),
    Actual := TO_DINT(ShapePublisher.Ring[1].ReasonCode), Message := 'reason carried');
TEST_FINISHED();
END_METHOD

METHOD Accepts_fixed_vocabulary
VAR
    i : INT;
    kind : E_HostEventKind;
END_VAR
TEST('Accepts_fixed_vocabulary');
FOR i := 1 TO 10 DO
    kind := i;
    AssertTrue(Condition := VocabularyPublisher.Emit(Kind := kind,
        StationPath := 'Root', PartUid := '', Subject := '', Value := '', Verdict := E_Verdict.NONE,
        ReasonCode := E_Reason.NONE), Message := 'fixed event kind accepted');
END_FOR
AssertEquals_INT(Expected := 10, Actual := VocabularyPublisher.Count,
    Message := 'exact fixed vocabulary emitted');
TEST_FINISHED();
END_METHOD

METHOD Ring_is_bounded
VAR
    i : INT;
END_VAR
TEST('Ring_is_bounded');
FOR i := 1 TO PL_Fraktal.MAX_HOST_EVENTS + 1 DO
    WrapPublisher.Emit(Kind := E_HostEventKind.MODE_CHANGED,
        StationPath := 'Root', PartUid := '', Subject := 'Mode',
        Value := '',
        Verdict := E_Verdict.NONE, ReasonCode := E_Reason.NONE);
END_FOR
AssertEquals_INT(Expected := PL_Fraktal.MAX_HOST_EVENTS, Actual := WrapPublisher.Count,
    Message := 'valid count saturates at the bound');
AssertEquals_INT(Expected := PL_Fraktal.MAX_HOST_EVENTS, Actual := WrapPublisher.Capacity,
    Message := 'published capacity derives from the owning PLC parameter');
AssertTrue(Condition := WrapPublisher.Wrapped, Message := 'overwrite is visible');
AssertEquals_INT(Expected := 1, Actual := WrapPublisher.RingHead,
    Message := 'bounded ring wraps deterministically');
TEST_FINISHED();
END_METHOD

END_FUNCTION_BLOCK

// ---- Fraktal_Tests/FB_InputCM_Tests.TcPOU
// Basic passive input types used to keep hardware-bound signals out of Units.
FUNCTION_BLOCK FB_InputCM_Tests EXTENDS TcUnit.FB_TestSuite
VAR
    _input : FB_DigitalInputCM;
    _air : FB_AirPressureMonitorCM;
    _inputHal : ST_DigitalInputHal;
    _airHal : ST_AirPressureHal;
    _inputIdentity, _lowIdentity, _operatingIdentity : ST_IoPointIdentity;
    _d : ST_Diagnostic;
    _wired : BOOL;
END_VAR

IF NOT _wired THEN
    _input.Setup(Name := 'Test.PartPresent', HalRef := _inputHal,
        DisplayNameKey := 'project.module.partPresentSensor.name',
        DescriptionKey := 'project.module.partPresentSensor.description');
    _inputIdentity.Tag := '_101B601'; _inputIdentity.Address := 'EL1809 Ch12';
    _input.ConfigureIoIdentity(Identity := _inputIdentity);
    _air.Setup(Name := 'Test.Air', HalRef := _airHal);
    // Deterministic qualification in the test runtime, set through the registered
// §3.10.2 capability rather than by touching the module's retained data: that
// path is the only one a station has, so the test uses it too.
_air.M_ApplyConfigWrite(Scope := 'Test.Air', WriteKey := 'airPressure.conflictTime',
    Revision := 1, TextValue := '0', RootReady := TRUE);
    _lowIdentity.Tag := '_000MB085A_2'; _lowIdentity.Address := 'EL1809 Ch10';
    _operatingIdentity.Tag := '_000MB085A_4'; _operatingIdentity.Address := 'EL1809 Ch11';
    _air.ConfigureIoIdentity(LowSensor := _lowIdentity, OperatingSensor := _operatingIdentity);
    _inputHal.Quality := TRUE; _airHal.Quality := TRUE;
    _wired := TRUE;
ELSE
    ;
END_IF
Digital_input_publishes_semantic_value_and_identity();
Air_monitor_derives_pressure_and_faults_on_conflict();

METHOD Digital_input_publishes_semantic_value_and_identity
TEST('Digital_input_publishes_semantic_value_and_identity');
_inputHal.Value := TRUE;
_input();
AssertTrue(Condition := _input.OutImm.Value, Message := 'HAL value published');
AssertEquals_STRING(Expected := '_101B601', Actual := _input.OutImm.IoTag,
    Message := 'physical identity is injected, not embedded in the type');
// §7.1: the display name is the instance's, the type key is the type's.
AssertEquals_STRING(Expected := 'project.module.partPresentSensor.name',
    Actual := _input.Status.DisplayNameKey, Message := 'display key is set per instance');
AssertEquals_STRING(Expected := 'std.moduleType.digitalInput', Actual := _input.Status.TypeKey,
    Message := 'type key is fixed by the type, whatever the instance is called');
TEST_FINISHED();
END_METHOD

METHOD Air_monitor_derives_pressure_and_faults_on_conflict
TEST('Air_monitor_derives_pressure_and_faults_on_conflict');
_airHal.LowPressure := FALSE; _airHal.OperatingPressure := TRUE;
_air();
AssertTrue(Condition := _air.OutImm.PressureOk,
    Message := 'operating threshold with low switch clear is ready');
_airHal.LowPressure := TRUE; _airHal.OperatingPressure := TRUE;
_air();
_d := _air.GetFaultSummary();
AssertEquals_DWORD(Expected := TO_DWORD(PL_ModuleReasons.AIR_SWITCH_CONFLICT),
    Actual := _air.ErrorID, Message := 'contradictory switches use registered type reason');
AssertEquals_STRING(Expected := '_000MB085A_2 / _000MB085A_4', Actual := _d.IoTag,
    Message := 'both implicated electrical tags are preserved');
TEST_FINISHED();
END_METHOD

END_FUNCTION_BLOCK

// ---- Fraktal_Tests/FB_ConfigWrite_Tests.TcPOU
// Core §3.8b/§3.10.2 under test: a module declares its own editable values, the
// root's walk publishes them as complete capabilities and carries writes back to
// the owner, and everything the owner did not agree to is refused without
// changing a byte. The pair FB_ProbeConfigUnit/FB_ProbeConfigCM deliberately
// contains no routing code — if these pass, a new module type needs none either.
FUNCTION_BLOCK FB_ConfigWrite_Tests EXTENDS TcUnit.FB_TestSuite
VAR
    _u : FB_ProbeConfigUnit;
    _init : BOOL;
    _setupOk : BOOL;
    _pager : FB_ConfigPager;
    _page : ST_ConfigPage;
    _found : ST_ConfigEntry;
    _dup : FB_ProbeConfigCM;
    _dupOk : BOOL;
END_VAR

